(* Logix 5000 project; controller PBS_Perfusion vendor 1 type 14 code 217 rev 32.14; software revision 32.03; part 8 of 27 *)
(* tags used below, declared in another part *)
   Inp : BOOL;   // Alarm Condition Input 1=Alarm
   Inp_OoS : ALIAS FOR Com_AE.2;   // 1=Out of Service (from object's P_CmdSrc)
   Cfg_Exists : BOOL;   // 1=Alarm configured to exist, 0=Does not exist, don't scan
   Cfg_ResetReqd : BOOL;   // 1=Latched Alarm, a Reset is required to clear this Alarm
   Cfg_AckReqd : BOOL;   // 1=Acknowledge required for this Alarm
   Cfg_AllowShelve : BOOL;   // 1=Allow Operator to Shelve this Alarm
   Cfg_AllowDisable : BOOL;   // 1=Allow Maintenance to Disable this Alarm
   Cfg_Severity : DINT;   // Alarm Severity: 1..250=Low, 251..500=Medium, 501..750=High, 751..1000=Urgent
   Cfg_AlmMinOnT : DINT;   // Minimum time Alm output stays on (sec)
   PCfg_AllowExist : BOOL;   // 1=Alarm can be configured to exist, 0=other configs make alarm meaningless
   PCmd_Ack : BOOL;   // Program Command to Acknowledge alarm
   PCmd_Suppress : BOOL;   // Program Command to Suppress by Design (inhibits new alarm)
   PCmd_Unsuppress : BOOL;   // Program Command to Unsuppress (allows new alarm)
   PCmd_Unshelve : BOOL;   // Program Command to Unshelve (e.g., on shift change)
   Alm : ALIAS FOR Com_AE.0;   // Alarm output 1=In Alarm
   Ack : ALIAS FOR Com_AE.1;   // Alarm acknowledged status: 1=Ack rcvd
   Shelved : ALIAS FOR Com_AE.3;   // 1=Alarm has been Shelved by Operator (inhibits new alarm)
   Suppressed : ALIAS FOR Com_AE.6;   // 1=Alarm has been Suppressed by Program (inhibits new alarm)
   Disabled : ALIAS FOR Com_AE.9;   // 1=Alarm has been Disabled by Maintanance (inhibits new alarm)
   P_Alarm : BOOL;   // Unique Parameter Name for auto - discovery
   Wrk_Suppressed : BOOL;   // Internal Alarm Suppressed Status
   Com_AE : INT;   // Communication with HMI / Alarm/Event Server (see bit descriptions)
   OCmd_Unshelve : BOOL;   // Operator Command to Unshelve alarm (allows new alarm)
   OCmd_Shelve : BOOL;   // Operator Command to Shelve Alarm (inhibits new alarm)
   OCmd_Ack : BOOL;   // Operator Command to Acknowledge alarm
   MCmd_Enable : BOOL;   // Maintenance Command to Enable alarm (allows new alarm)
   MCmd_Disable : BOOL;   // Maintenance Command to Disable alarm (inhibits new alarm)
   ONS : DINT[3];
   REAL : DINT;
(* P_Alarm, continued *)

ROUTINE Prescan   (* ladder *)
// Clear "lurking" Commands
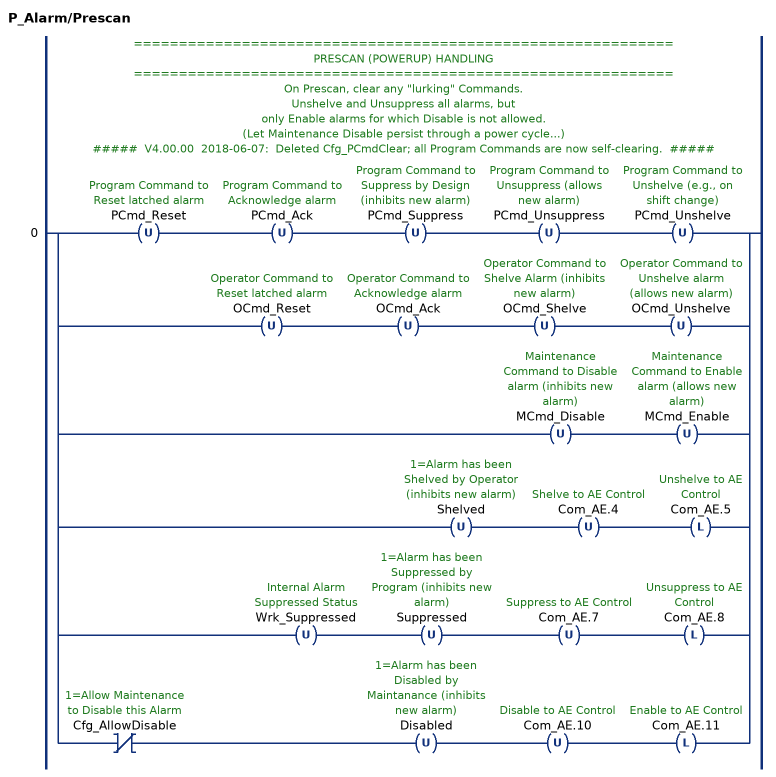
   // ============================================================
   // PRESCAN (POWERUP) HANDLING
   // ============================================================
   // On Prescan, clear any "lurking" Commands.
   // Unshelve and Unsuppress all alarms, but
   // only Enable alarms for which Disable is not allowed.
   // (Let Maintenance Disable persist through a power cycle...)
   // #####  V4.00.00  2018-06-07:  Deleted Cfg_PCmdClear; all Program Commands are now self-clearing.  #####
   0: [OTU(PCmd_Reset) OTU(PCmd_Ack) OTU(PCmd_Suppress) OTU(PCmd_Unsuppress) OTU(PCmd_Unshelve) ,OTU(OCmd_Reset) OTU(OCmd_Ack) OTU(OCmd_Shelve) OTU(OCmd_Unshelve) ,OTU(MCmd_Disable) OTU(MCmd_Enable) ,OTU(Shelved) OTU(Com_AE.4) OTL(Com_AE.5) ,OTU(Wrk_Suppressed) OTU(Suppressed) OTU(Com_AE.7) OTL(Com_AE.8) ,XIO(Cfg_AllowDisable) OTU(Disabled) OTU(Com_AE.10) OTL(Com_AE.11) ];
END_ROUTINE
END_ADD_ON_INSTRUCTION

ADD_ON_INSTRUCTION P_AOut   (* revision 4.10 .01 Release, vendor Rockwell Automation, ExecutePrescan, ExecuteEnableInFalse *)
// Analog Output
// Revision note:
// See Instruction Help for a summary of changes, and see 4.10 Release Notes for details.
// Help:
// Copyright © Rockwell Automation, Inc.  All Rights Reserved.
// This Instruction controls an Analog Output and provides:
// *  Program and Operator entry of target CV in Engineering Units
// *  Ramping of Output CV to target at specified Rate of Change (EU/sec)
// *  Clamping of Output CV at configured minimum and maximum limits
// *  Scaling of Output CV from Engineering Units to Raw (I/O card) Units
// *  Monitoring of Interlock conditions which cause output to shed
// *  Configurable shed to HOLD or to configured value
// *  Monitoring of I/O communication faults
// *  Alarms for Interlock Trip, I/O Fault
// *  "Available" status for use by automation logic to know whether Output
//       can be controlled by other objects.
// Command Sources are arbitrated by a P_CmdSrc Add-On Instruction instance.
// Command Sources: Operator, Program, External, Override, Maintenance, Out of
// Service, Hand.  Alarms are provided by P_Alarm Add-On Instruction instances.
// SUMMARY OF CHANGES FROM PREVIOUS VERSION (4.10.00)
// See 4.10 Release Notes for details.
// * No changes, uprevved because P_CmdSrc 4.10.01 is used.
// PREVIOUS VERSION (4.00.00)
// See 4.10 Release Notes for details.
// * Changed Sts_Available to use input availability from interlocks.
// * Updated to P_CmdSrc V4.10.00.
// * Added Cfg_HasMoreObj
// SUMMARY OF CHANGES FROM PREVIOUS VERSION (3.5-11)
// See 4.00 Release Notes for details.
// * Changed Inf_ items to HMI_, and added Cfg_Area for security.
// * Added notify and unack count rollup for associated object(s).
// * Changed "Mode" to "Command Source" using P_CmdSrc 4.00.00.
// * Deleted Cfg_PCmdClear; all Program Commands are now self-clearing.
// * Aligned ready bit naming with command bit names.
// * Added unacked alarm count.
// * Added  configurable decimal places for display on HMI.
// * Corrected CV Rate of Change Limiting when one direction is unlimited.
// * All OCmds/MCmds and ORdys/MRdys are now Local Tags.
// * Added Sts_RdyAck and Sts_RdyReset for use by external objects.
VAR_INPUT
   Inp_Tieback : REAL; {visible}   // Tieback CV (in raw, Out_CV units) used in Hand or Init
   Inp_IntlkOK : BOOL := 1; {visible}   // 1=Interlocks OK, Analog Output can be set
   Inp_NBIntlkOK : BOOL := 1; {visible}   // 1=Non-Bypassable Interlocks OK, Analog Output can be set
   Inp_IntlkAvail : BOOL;   // 1 = Interlock Availibility OK
   Inp_IOFault : BOOL;   // Input Communication Status 0=OK, 1=fail
   Inp_Sim : BOOL;   // 1=I/O are being simulated, set output CV to 0, ignore I/O Fault
   Inp_Hand : ALIAS FOR CmdSrc.Inp_Hand; {visible}
   Inp_Ovrd : ALIAS FOR CmdSrc.Inp_Ovrd; {visible}
   Inp_OvrdCV : REAL; {visible}   // CV target in Override Mode
   Inp_ExtInh : ALIAS FOR CmdSrc.Inp_ExtInh;
   Inp_Reset : BOOL;   // 1=Reset shed latches and cleared alarms
   Cfg_ShedHold : BOOL;   // 1=Hold Output on Interlock, 0=Go to Cfg_IntlkCV
   Cfg_SkipRoCLim : BOOL;   // 1=Skip RoC Limiting in Intlk, Maint, Ovrd
   Cfg_SetTrack : BOOL := 1;   // 1=PSets track OSets in Oper, OSets track PSets in Prog, 0=no tracking
   Cfg_SetTrackOvrdHand : BOOL;   // 1=Prog/Oper Settings track Override/Hand CV
   Cfg_HasIntlkObj : BOOL;   // 1=Tells HMI a P_Intlk is connected to Inp_Intlk
   Cfg_HasMoreObj : BOOL;   // 1=Tells HMI an object with more info is available
   Cfg_HasCVNav : BOOL;   // 1=Tells HMI to enable navigation to a connected CV object
   Cfg_OvrdIntlk : BOOL;   // 1=Override ignores Bypassable Intlk; 0=always use Intlk
   Cfg_ShedOnIOFault : BOOL := 1;   // 1=Stop Motor and Alarm on I/O Fault; 0=Alarm only on I/O Fault
   Cfg_DecPlcs : DINT := 2;   // Number of decimal places for CV display (0..6)
   Cfg_HasIntlkTripAlm : ALIAS FOR IntlkTrip.Cfg_Exists;   // 1=Interlock Trip Alarm exists and will be checked
   Cfg_HasIOFaultAlm : ALIAS FOR IOFault.Cfg_Exists;   // 1=I/O Fault Alarm exists and will be checked
   Cfg_IntlkTripResetReqd : ALIAS FOR IntlkTrip.Cfg_ResetReqd;   // 1=Reset required to clear Interlock Trip Alarm
   Cfg_IOFaultResetReqd : ALIAS FOR IOFault.Cfg_ResetReqd;   // 1=Reset required to clear I/O Fault Alarm
   Cfg_IntlkTripAckReqd : ALIAS FOR IntlkTrip.Cfg_AckReqd;   // 1=Acknowledge required for Interlock Trip Alarm
   Cfg_IOFaultAckReqd : ALIAS FOR IOFault.Cfg_AckReqd;   // 1=Acknowledge required for I/O Fault Alarm
   Cfg_IntlkTripSeverity : ALIAS FOR IntlkTrip.Cfg_Severity;   // Interlock Trip Alarm Severity: 1..250=Low, 251..500=Medium, 501..750=High, 751..1000=Urgent
   Cfg_IOFaultSeverity : ALIAS FOR IOFault.Cfg_Severity;   // I/O Fault Alarm Severity: 1..250=Low, 251..500=Medium, 501..750=High, 751..1000=Urgent
   Cfg_MinCV : REAL;   // Minimum CV (in EU, for limiting)
   Cfg_MaxCV : REAL := 100.0;   // Maximum CV (in EU, for limiting)
   Cfg_CVRoCLimInc : REAL;   // CV Rate of Change Limit, Increasing, (EU/sec, 0=unlimited)
   Cfg_CVRoCLimDec : REAL;   // CV Rate of Change Limit, Decreasing, (EU/sec, 0=unlimited)
   Cfg_IntlkCV : REAL;   // CV Target when interlocked (if not Cfg_ShedHold) (EU)
   Cfg_CVEUMin : REAL;   // CV Minimum in Engineering Units (for scaling)
   Cfg_CVEUMax : REAL := 100.0;   // CV Maximum in Engineering Units (for scaling)
   Cfg_CVRawMin : REAL;   // CV Minimum in I/O (raw) Units (for scaling)
   Cfg_CVRawMax : REAL := 100.0;   // CV Maximum in I/O (raw) Units (for scaling)
   Cfg_MaxInactiveCV : REAL;   // When Val_CVOut is greater than this value (in CV EU) set Sts_Active (for HMI)
   PSet_CV : REAL;   // Program Setting of Controlled Variable (output) (in EU)
   PSet_Owner : DINT;   // Program Owner Request ID (non-zero) or Release (zero)
   XSet_CV : REAL;   // External Setting of Controlled Variable (output) (in EU)
   PCmd_Prog : ALIAS FOR CmdSrc.PCmd_Prog;
   PCmd_Oper : ALIAS FOR CmdSrc.PCmd_Oper;
   PCmd_Lock : ALIAS FOR CmdSrc.PCmd_Lock;
   PCmd_Unlock : ALIAS FOR CmdSrc.PCmd_Unlock;
   PCmd_Normal : ALIAS FOR CmdSrc.PCmd_Normal;
   PCmd_Reset : BOOL;   // Program Command to reset shed latches and cleared alarms
   PCmd_IntlkTripAck : ALIAS FOR IntlkTrip.PCmd_Ack;   // Program Command to Acknowledge Interlock Trip Alarm
   PCmd_IntlkTripSuppress : ALIAS FOR IntlkTrip.PCmd_Suppress;   // Program Command to Suppress Interlock Trip Alarm
   PCmd_IntlkTripUnsuppress : ALIAS FOR IntlkTrip.PCmd_Unsuppress;   // Program Command to Unsuppress Interlock Trip Alarm
   PCmd_IntlkTripUnshelve : ALIAS FOR IntlkTrip.PCmd_Unshelve;   // Program Command to Unshelve Interlock Trip Alarm
   PCmd_IOFaultAck : ALIAS FOR IOFault.PCmd_Ack;   // Program Command to Acknowledge I/O Fault Alarm
   PCmd_IOFaultSuppress : ALIAS FOR IOFault.PCmd_Suppress;   // Program Command to Suppress I/O Fault Alarm
   PCmd_IOFaultUnsuppress : ALIAS FOR IOFault.PCmd_Unsuppress;   // Program Command to Unsuppress I/O Fault Alarm
   PCmd_IOFaultUnshelve : ALIAS FOR IOFault.PCmd_Unshelve;   // Program Command to Unshelve I/O Fault Alarm
   MCmd_Rel : ALIAS FOR CmdSrc.MCmd_Rel;
   OCmd_Unlock : ALIAS FOR CmdSrc.OCmd_Unlock;
   XCmd_Acq : ALIAS FOR CmdSrc.XCmd_Acq;
   XCmd_Rel : ALIAS FOR CmdSrc.XCmd_Rel;
   XCmd_Reset : BOOL;   // External Command to reset shed latches and cleared alarms
END_VAR
VAR_OUTPUT
   Out_CV : REAL; {access Read Only, visible}   // CV Output in Raw (I/O Card) Units
   Val_CVSet : REAL; {access Read Only, visible}   // Value of selected CV Setting (before rate limiting, in EU)
   Val_CVOut : REAL; {access Read Only, visible}   // Value of CV Output (after rate limiting) (in EU)
   Val_CVEUMin : REAL; {access Read Only}   // Minimum of scaled range = MIN (Cfg_CVEUMin, Cfg_CVEUMax)
   Val_CVEUMax : REAL := 100.0; {access Read Only}   // Maximum of scaled range = MAX (Cfg_CVEUMin, Cfg_CVEUMax)
   SrcQ_IO : DINT; {access Read Only}   // Source and Quality of primary I/O (enumeration)
   SrcQ : DINT; {access Read Only}   // Source and Quality of primary Val/Sts (enumeration)
   Val_Sts : DINT; {access Read Only}   // 0=AtTgt 1=RampDn 2=RampUp 3=ClampMin 4=ClampMax
   Val_Fault : DINT; {access Read Only}   // Device Fault Status 0=none, 32=I/OFault, 34=CfgErr
   Val_NotifyAll : DINT; {access Read Only}   // Highest Alarm prio and ack status this object + channel (enum)
   Val_UnackAlmC : DINT; {access Read Only}   // Count of Unacknowledged Alarms
   Val_Owner : DINT; {access Read Only}   // Current Object Owner ID (0=not owned)
   Sts_Ramping : BOOL; {access Read Only}   // 1=CV is ramping to target
   Sts_Clamped : BOOL; {access Read Only}   // 1=CV Set is clamped at CVMin or CVMax
   Sts_SkipRoCLim : BOOL; {access Read Only}   // 1=Rate of Change Limiting was skipped this scan (Maint, Ovrd, Intlk, Hand)
   Sts_Active : BOOL; {access Read Only}   // 1=CV is greater than Cfg_MaxInactiveCV, show graphic symbol as "active"
   Sts_Available : BOOL; {access Read Only}   // 1=Analog Output available for control by automation (Prog)
   Sts_Bypass : BOOL; {access Read Only}   // 1=Bypassable Interlocks are Bypassed
   Sts_BypActive : BOOL; {access Read Only}   // 1=Bypassing Active (Bypassed or Maintenance)
   Sts_NotRdy : BOOL; {access Read Only}   // 1=Device Not Ready, see detail bits for reason
   Nrdy_CfgErr : BOOL; {access Read Only}   // 1=Device Not Ready: Configuration Error
   Nrdy_Intlk : BOOL; {access Read Only}   // 1=Device Not Ready: Interlock Not OK
   Nrdy_IOFault : BOOL; {access Read Only}   // 1=Device Not Ready: I/O Fault (Shed Requires Reset)
   Nrdy_OoS : BOOL; {access Read Only}   // 1=Device Not Ready: Device is Out of Service
   Sts_MaintByp : BOOL; {access Read Only}   // 1=Device has a Maintenance Bypass function active
   Sts_AlmInh : BOOL; {access Read Only}   // 1=One or more Alarms Shelved, Disabled or Suppressed
   Sts_Err : BOOL; {access Read Only, visible}   // 1=Error in Config: see detail bits for reason
   Err_Limit : BOOL; {access Read Only}   // 1=Error in Config: CV Limits swapped
   Err_EU : BOOL; {access Read Only}   // 1=Error in Config: Scaled CV EU Min = Max
   Err_Raw : BOOL; {access Read Only}   // 1=Error in Config: Raw Output Scaling Min = Max
   Err_Alarm : BOOL; {access Read Only}   // 1=Error in Config: Alarm Min On Time, Shelf Time, Severity
   Sts_Hand : ALIAS FOR CmdSrc.Sts_Hand; {access Read Only, visible}
   Sts_OoS : ALIAS FOR CmdSrc.Sts_OoS; {access Read Only, visible}
   Sts_Maint : ALIAS FOR CmdSrc.Sts_Maint; {access Read Only, visible}
   Sts_Ovrd : ALIAS FOR CmdSrc.Sts_Ovrd; {access Read Only, visible}
   Sts_Ext : ALIAS FOR CmdSrc.Sts_Ext; {access Read Only, visible}
   Sts_Prog : ALIAS FOR CmdSrc.Sts_Prog; {access Read Only, visible}
   Sts_ProgLocked : ALIAS FOR CmdSrc.Sts_ProgLocked; {access Read Only}
   Sts_Oper : ALIAS FOR CmdSrc.Sts_Oper; {access Read Only, visible}
   Sts_OperLocked : ALIAS FOR CmdSrc.Sts_OperLocked; {access Read Only}
   Sts_Normal : ALIAS FOR CmdSrc.Sts_Normal; {access Read Only}
   Sts_ExtReqInh : ALIAS FOR CmdSrc.Sts_ExtReqInh; {access Read Only}
   Sts_ProgReqInh : ALIAS FOR CmdSrc.Sts_ProgReqInh; {access Read Only}
   Sts_MAcqRcvd : ALIAS FOR CmdSrc.Sts_MAcqRcvd; {access Read Only}
   Sts_RdyReset : ALIAS FOR ORdy_Reset; {access Read Only}   // 1=A latched alarm or shed condition is ready to be reset
   Sts_RdyAck : BOOL; {access Read Only}   // 1=An alarm is ready to be acknowledged
   Sts_IntlkTrip : ALIAS FOR IntlkTrip.Inp;   // 1=Status: CV held or forced by interlock NOT OK (1-shot)
   Alm_IntlkTrip : ALIAS FOR IntlkTrip.Alm;   // 1=Alarm: CV held or forced by interlock NOT OK
   Ack_IntlkTrip : ALIAS FOR IntlkTrip.Ack;   // 1=Interlock Trip Alarm has been acknowledged
   Sts_IntlkTripDisabled : ALIAS FOR IntlkTrip.Disabled;   // 1=Interlock Trip Alarm has been Disabled by Maintenance
   Sts_IntlkTripShelved : ALIAS FOR IntlkTrip.Shelved;   // 1=Interlock Trip Alarm has been Shelved by Operator
   Sts_IntlkTripSuppressed : ALIAS FOR IntlkTrip.Suppressed;   // 1=Interlock Trip Alarm has been Suppressed by Program
   Sts_IOFault : ALIAS FOR IOFault.Inp;   // 1=I/O Fault Status (0=OK, 1=Bad)
   Alm_IOFault : ALIAS FOR IOFault.Alm;   // 1=I/O Fault Alarm
   Ack_IOFault : ALIAS FOR IOFault.Ack;   // 1=I/O Fault Alarm has been acknowledged
   Sts_IOFaultDisabled : ALIAS FOR IOFault.Disabled;   // 1=I/O Fault Alarm has been Disabled by Maintenance
   Sts_IOFaultShelved : ALIAS FOR IOFault.Shelved;   // 1=I/O Fault Alarm has been Shelved by Operator
   Sts_IOFaultSuppressed : ALIAS FOR IOFault.Suppressed;   // 1=I/O Fault Alarm has been Suppressed by Program
   MRdy_Rel : ALIAS FOR CmdSrc.MRdy_Rel; {access Read Only}
   ORdy_Unlock : ALIAS FOR CmdSrc.ORdy_Unlock; {access Read Only}
   P_AOut : BOOL;   // Unique Parameter Name for auto - discovery
END_VAR
VAR
   CmdSrc : P_CmdSrc := (Cfg_HasOper := 1, Cfg_HasOperLocked := 1, Cfg_HasProg := 1, Cfg_HasProgLocked := 1, Cfg_HasMaint := 1, Cfg_HasMOoS := 1, Cfg_OvrdOverLock := 1, Sts_bSrc := 1);   // Control / Command Source Selection
   IOFault : P_Alarm := (Cfg_AckReqd := 1, Cfg_AllowShelve := 1, Cfg_AllowDisable := 1, Cfg_Severity := 1000, Cfg_AlmMinOnT := 5, PCfg_AllowExist := 1, Ack := 1);   // I/O Fault Alarm
   IntlkTrip : P_Alarm := (Cfg_AckReqd := 1, Cfg_AllowShelve := 1, Cfg_AllowDisable := 1, Cfg_Severity := 500, Cfg_AlmMinOnT := 5, PCfg_AllowExist := 1, Ack := 1);   // Interlock Trip Alarm
   Cfg_Tag : STRING_20 := 'P_AOut';   // Tagname for display on HMI
   Cfg_Label : STRING_20 := 'Analog Output';   // Label for graphic symbol displayed on HMI
   Cfg_Desc : STRING_40 := 'Analog Output';   // Description for display on HMI
   Wrk_Notify : DINT; {access None}   // Buffer for building Val_Notify
   Wrk_Bypass : BOOL; {access None}   // Internal Bypassable Interlocks are Bypassed flag
   Cfg_EU : STRING_8 := '%';   // Engineering Units for display on HMI
   Wrk_CV : REAL; {access None}   // Working copy of Speed Reference (for limiting)
   Wrk_CVSet : REAL; {access None}   // Final selected CV to feed to RoC Limiter
   Wrk_CVOut : REAL; {access None}   // Wroking value of CV after Rate Limiting
   Wrk_IntlkTripONS : BOOL; {access None}   // Interlock Tripped This Scan
   Wrk_ScanTime : REAL; {access None}   // Seconds since previous scan
   Wrk_StepInc : REAL; {access None}   // Amount to change CVOut this scan for increase rate limiting
   Wrk_ScanT : TIMER := (PRE := 2147483647); {access None}   // Scan Timer (milliseconds, always runs)
   Wrk_SelCVDINT : DINT; {access None}   // Selected CV check for Infinite or Non A Number
   HMI_Tab : SINT;   // Tab to display (FTView ME)
   Val_Notify : SINT; {access Read Only}   // Current Alarm Level and Acknowledgement (enumeration)
   Wrk_Sts : DINT; {access None}   // Buffer for building Val_Sts
   Wrk_Fault : DINT; {access None}   // Buffer for building Val_Fault
   Wrk_SrcQ : DINT; {access None}   // Register for building Source / Quality enumeration
   HMI_Type : STRING_16 := 'P_AOut'; {access Read Only}   // Must contain AOI name, used for HMI and Information S/W
   Wrk_StepDec : REAL; {access None}   // Amount to change CVOut this scan for decrease rate limiting
   HMI_Lib : STRING_12 := 'RA-BAS'; {access Read Only}   // Display Library for Faceplate call-up
   Cfg_CVNavTag : STRING_NavTag;   // Tagname for destination of CV Navigation button
   Wrk_ShedIntlkCV : BOOL; {access None}   // Output CV being held at Interlock value
   Wrk_ShedHold : BOOL; {access None}   // Output CV being held at last good value
   Cfg_Area : STRING_Area := 'area01';   // Process Area for security
   Wrk_UnackAlmC : DINT; {access None}   // Buffer for building Val_UnackAlmC
   ORdy_CV : BOOL; {access Read Only}   // 1=Ready for OSet_CV (enables data entry field)
   ORdy_ResetAckAll : BOOL; {access Read Only}   // 1=Ready for OCmd_ResetAckAll (enables HMI button)
   ORdy_Reset : BOOL; {access Read Only}   // 1=Ready for OCmd_Reset (enables HMI button)
   MRdy_Check : BOOL; {access Read Only}   // 1=Ready for MCmd_Check (enables HMI button)
   MRdy_Bypass : BOOL; {access Read Only}   // 1=Ready for MCmd_Bypass (enables HMI button)
   OCmd_ResetAckAll : BOOL;   // Operator Command to Reset all Alarms and latched Shed conditions
   OCmd_Reset : BOOL;   // Oper Cmd to reset shed latches and cleared alarms
   MCmd_Check : BOOL;   // Maintenance Command to Check (not bypass) all Interlocks
   MCmd_Bypass : BOOL;   // Maintenance Command to Bypass all Bypassable Interlocks
   OSet_CV : REAL;   // Operator Setting of Controlled Variable (output) (in EU)
END_VAR

ROUTINE EnableInFalse   (* ladder *)
// Out of Service is asserted, Output OFF (zero), Alarms inhibited.
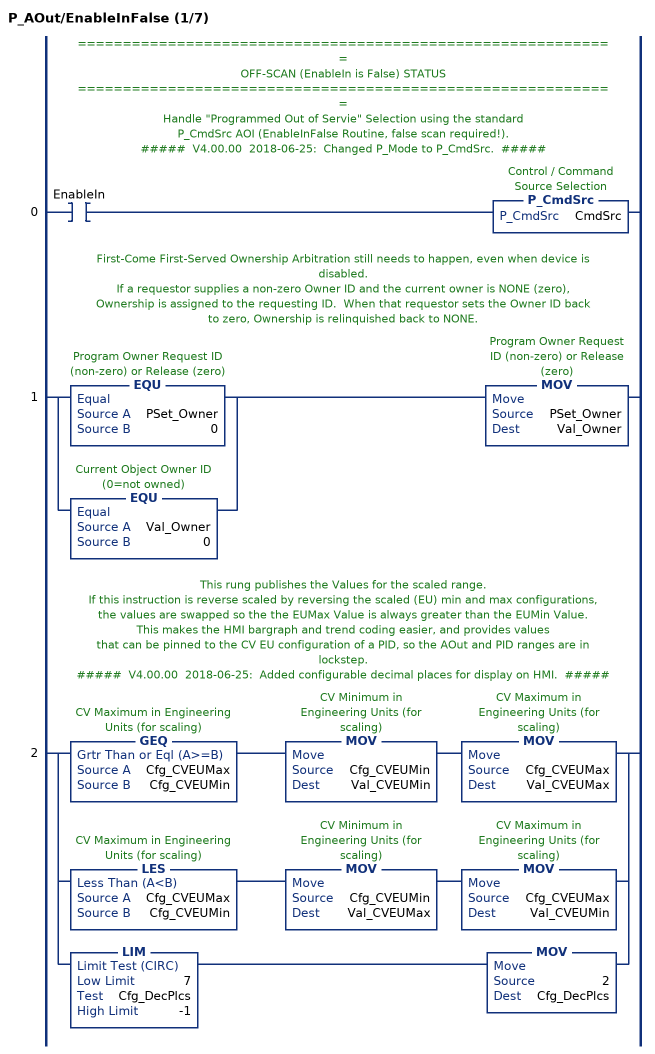
   // ============================================================
   // OFF-SCAN (EnableIn is False) STATUS
   // ============================================================
   // Handle "Programmed Out of Servie" Selection using the standard
   // P_CmdSrc AOI (EnableInFalse Routine, false scan required!).
   // #####  V4.00.00  2018-06-25:  Changed P_Mode to P_CmdSrc.  #####
   0: XIC(EnableIn)P_CmdSrc(CmdSrc);
   // First-Come First-Served Ownership Arbitration still needs to happen, even when device is disabled.
   // If a requestor supplies a non-zero Owner ID and the current owner is NONE (zero),
   // Ownership is assigned to the requesting ID.  When that requestor sets the Owner ID back
   // to zero, Ownership is relinquished back to NONE.
   1: [EQU(PSet_Owner,0) ,EQU(Val_Owner,0) ]MOV(PSet_Owner,Val_Owner);
   // This rung publishes the Values for the scaled range.
   // If this instruction is reverse scaled by reversing the scaled (EU) min and max configurations,
   // the values are swapped so the the EUMax Value is always greater than the EUMin Value.
   // This makes the HMI bargraph and trend coding easier, and provides values
   // that can be pinned to the CV EU configuration of a PID, so the AOut and PID ranges are in lockstep.
   // #####  V4.00.00  2018-06-25:  Added configurable decimal places for display on HMI.  #####
   2: [GEQ(Cfg_CVEUMax,Cfg_CVEUMin) MOV(Cfg_CVEUMin,Val_CVEUMin) MOV(Cfg_CVEUMax,Val_CVEUMax) ,LES(Cfg_CVEUMax,Cfg_CVEUMin) MOV(Cfg_CVEUMin,Val_CVEUMax) MOV(Cfg_CVEUMax,Val_CVEUMin) ,LIM(7,Cfg_DecPlcs,-1) MOV(2,Cfg_DecPlcs) ];
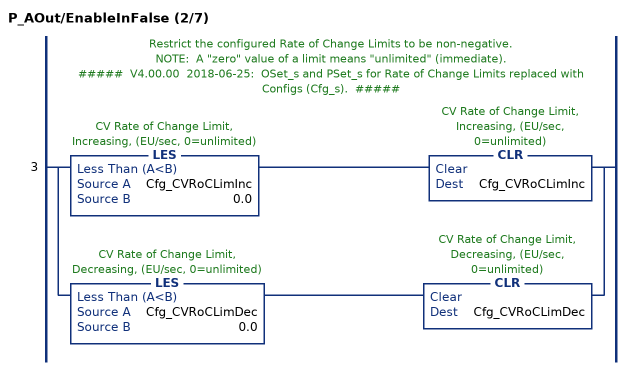
   // Restrict the configured Rate of Change Limits to be non-negative.
   // NOTE:  A "zero" value of a limit means "unlimited" (immediate).
   // #####  V4.00.00  2018-06-25:  OSet_s and PSet_s for Rate of Change Limits replaced with Configs (Cfg_s).  #####
   3: [LES(Cfg_CVRoCLimInc,0.0) CLR(Cfg_CVRoCLimInc) ,LES(Cfg_CVRoCLimDec,0.0) CLR(Cfg_CVRoCLimDec) ];
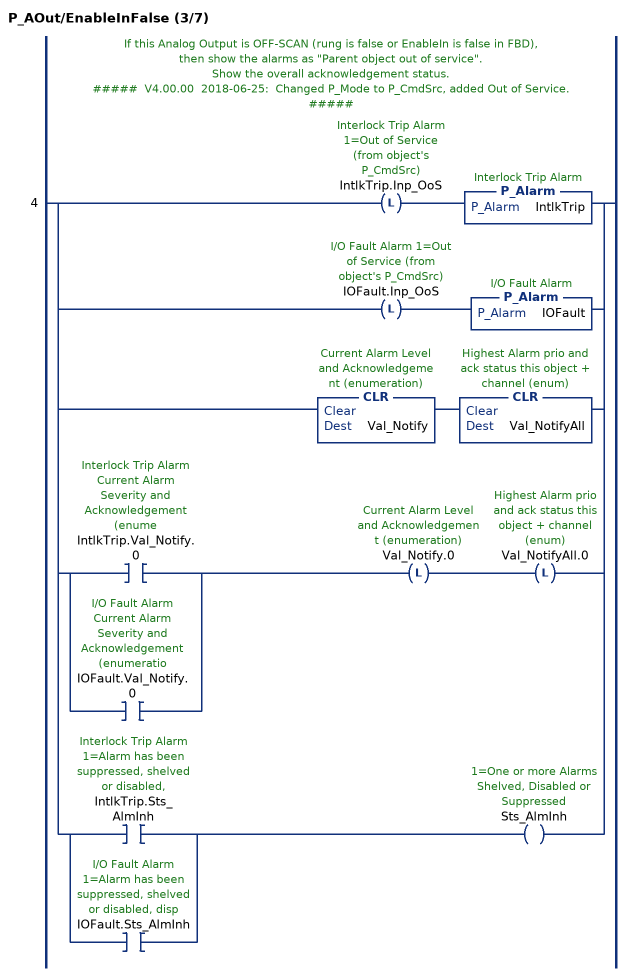
   // If this Analog Output is OFF-SCAN (rung is false or EnableIn is false in FBD),
   // then show the alarms as "Parent object out of service".
   // Show the overall acknowledgement status.
   // #####  V4.00.00  2018-06-25:  Changed P_Mode to P_CmdSrc, added Out of Service.  #####
   4: [OTL(IntlkTrip.Inp_OoS) P_Alarm(IntlkTrip) ,OTL(IOFault.Inp_OoS) P_Alarm(IOFault) ,CLR(Val_Notify) CLR(Val_NotifyAll) ,[XIC(IntlkTrip.Val_Notify.0) ,XIC(IOFault.Val_Notify.0) ] OTL(Val_Notify.0) OTL(Val_NotifyAll.0) ,[XIC(IntlkTrip.Sts_AlmInh) ,XIC(IOFault.Sts_AlmInh) ] OTE(Sts_AlmInh) ];
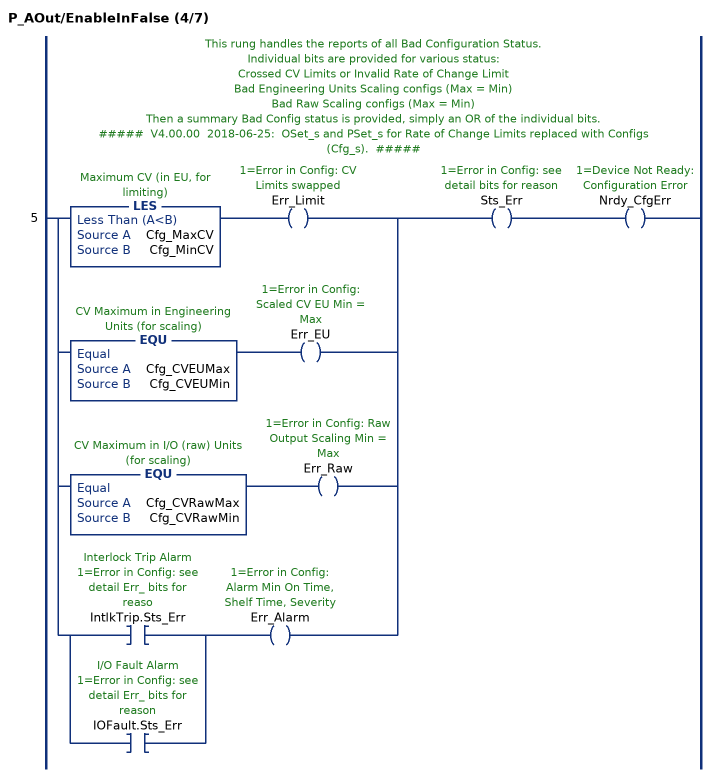
   // This rung handles the reports of all Bad Configuration Status.
   // Individual bits are provided for various status:
   // Crossed CV Limits or Invalid Rate of Change Limit
   // Bad Engineering Units Scaling configs (Max = Min)
   // Bad Raw Scaling configs (Max = Min)
   // Then a summary Bad Config status is provided, simply an OR of the individual bits.
   // #####  V4.00.00  2018-06-25:  OSet_s and PSet_s for Rate of Change Limits replaced with Configs (Cfg_s).  #####
   5: [LES(Cfg_MaxCV,Cfg_MinCV) OTE(Err_Limit) ,EQU(Cfg_CVEUMax,Cfg_CVEUMin) OTE(Err_EU) ,EQU(Cfg_CVRawMax,Cfg_CVRawMin) OTE(Err_Raw) ,[XIC(IntlkTrip.Sts_Err) ,XIC(IOFault.Sts_Err) ] OTE(Err_Alarm) ]OTE(Sts_Err)OTE(Nrdy_CfgErr);
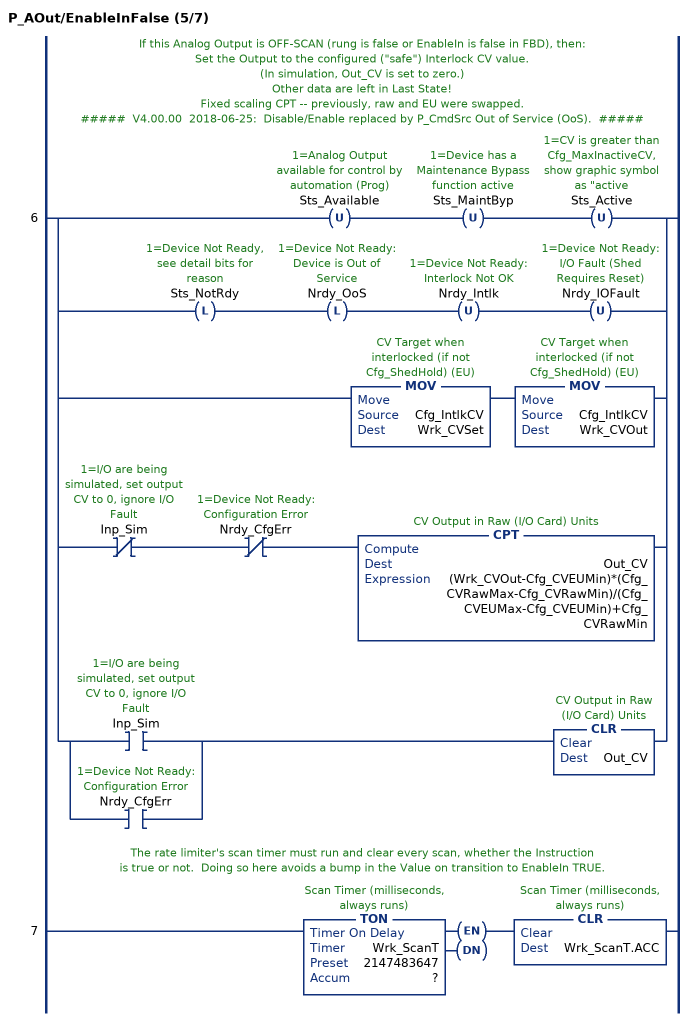
   // If this Analog Output is OFF-SCAN (rung is false or EnableIn is false in FBD), then:
   // Set the Output to the configured ("safe") Interlock CV value.
   // (In simulation, Out_CV is set to zero.)
   // Other data are left in Last State!
   // Fixed scaling CPT -- previously, raw and EU were swapped.
   // #####  V4.00.00  2018-06-25:  Disable/Enable replaced by P_CmdSrc Out of Service (OoS).  #####
   6: [OTU(Sts_Available) OTU(Sts_MaintByp) OTU(Sts_Active) ,OTL(Sts_NotRdy) OTL(Nrdy_OoS) OTU(Nrdy_Intlk) OTU(Nrdy_IOFault) ,MOV(Cfg_IntlkCV,Wrk_CVSet) MOV(Cfg_IntlkCV,Wrk_CVOut) ,XIO(Inp_Sim) XIO(Nrdy_CfgErr) CPT(Out_CV,(Wrk_CVOut-Cfg_CVEUMin)*(Cfg_CVRawMax-Cfg_CVRawMin)/(Cfg_CVEUMax-Cfg_CVEUMin)+Cfg_CVRawMin) ,[XIC(Inp_Sim) ,XIC(Nrdy_CfgErr) ] CLR(Out_CV) ];
   // The rate limiter's scan timer must run and clear every scan, whether the Instruction
   // is true or not.  Doing so here avoids a bump in the Value on transition to EnableIn TRUE.
   7: TON(Wrk_ScanT,?,?)CLR(Wrk_ScanT.ACC);
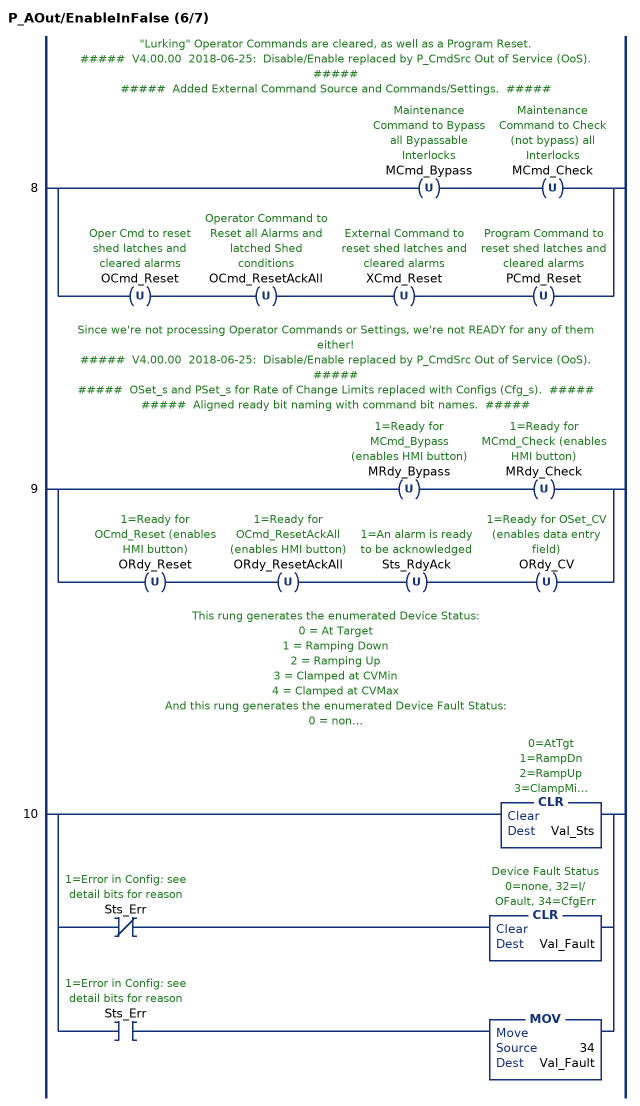
   // "Lurking" Operator Commands are cleared, as well as a Program Reset.
   // #####  V4.00.00  2018-06-25:  Disable/Enable replaced by P_CmdSrc Out of Service (OoS).  #####
   // #####  Added External Command Source and Commands/Settings.  #####
   8: [OTU(MCmd_Bypass) OTU(MCmd_Check) ,OTU(OCmd_Reset) OTU(OCmd_ResetAckAll) OTU(XCmd_Reset) OTU(PCmd_Reset) ];
   // Since we're not processing Operator Commands or Settings, we're not READY for any of them either!
   // #####  V4.00.00  2018-06-25:  Disable/Enable replaced by P_CmdSrc Out of Service (OoS).  #####
   // #####  OSet_s and PSet_s for Rate of Change Limits replaced with Configs (Cfg_s).  #####
   // #####  Aligned ready bit naming with command bit names.  #####
   9: [OTU(MRdy_Bypass) OTU(MRdy_Check) ,OTU(ORdy_Reset) OTU(ORdy_ResetAckAll) OTU(Sts_RdyAck) OTU(ORdy_CV) ];
   // This rung generates the enumerated Device Status:
   // 0 = At Target
   // 1 = Ramping Down
   // 2 = Ramping Up
   // 3 = Clamped at CVMin
   // 4 = Clamped at CVMax
   // And this rung generates the enumerated Device Fault Status:
   // 0 = none
   // 32 = I/O Fault
   // 34 = Configuration Error
   // #####  V4.00.00  2018-06-25:  Disable/Enable replaced by P_CmdSrc Out of Service (OoS).  #####
   10: [CLR(Val_Sts) ,XIO(Sts_Err) CLR(Val_Fault) ,XIC(Sts_Err) MOV(34,Val_Fault) ];
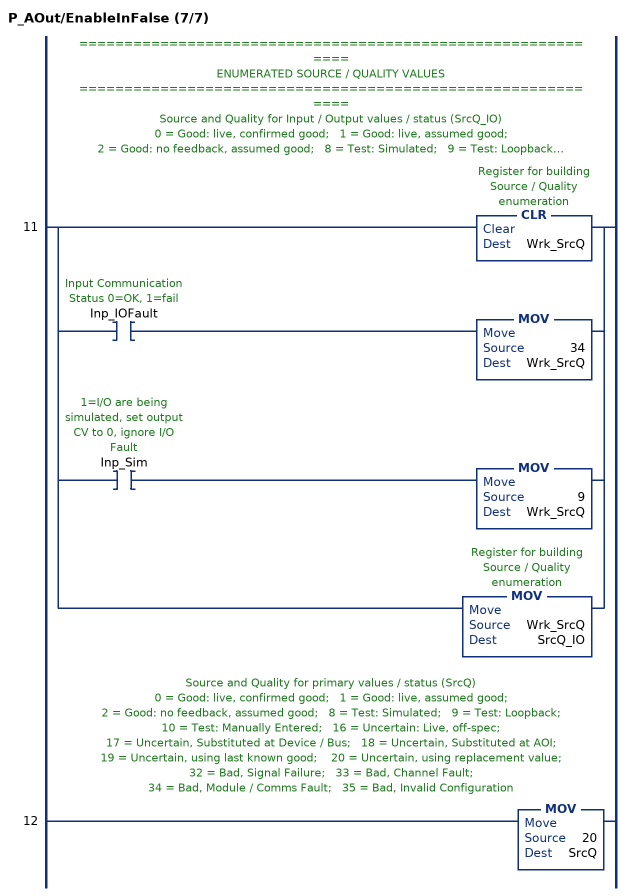
   // ============================================================
   // ENUMERATED SOURCE / QUALITY VALUES
   // ============================================================
   // Source and Quality for Input / Output values / status (SrcQ_IO)
   // 0 = Good: live, confirmed good;   1 = Good: live, assumed good;
   // 2 = Good: no feedback, assumed good;   8 = Test: Simulated;   9 = Test: Loopback;
   // 10 = Test: Manually Entered;   16 = Uncertain: Live, off-spec;
   // 17 = Uncertain, Substituted at Device / Bus;   18 = Uncertain, Substituted at AOI;
   // 19 = Uncertain, using last known good;    20 = Uncertain, using replacement value;
   // 32 = Bad, Signal Failure;   33 = Bad, Channel Fault;
   // 34 = Bad, Module / Comms Fault;   35 = Bad, Invalid Configuration
   11: [CLR(Wrk_SrcQ) ,XIC(Inp_IOFault) MOV(34,Wrk_SrcQ) ,XIC(Inp_Sim) MOV(9,Wrk_SrcQ) ,MOV(Wrk_SrcQ,SrcQ_IO) ];
   // Source and Quality for primary values / status (SrcQ)
   // 0 = Good: live, confirmed good;   1 = Good: live, assumed good;
   // 2 = Good: no feedback, assumed good;   8 = Test: Simulated;   9 = Test: Loopback;
   // 10 = Test: Manually Entered;   16 = Uncertain: Live, off-spec;
   // 17 = Uncertain, Substituted at Device / Bus;   18 = Uncertain, Substituted at AOI;
   // 19 = Uncertain, using last known good;    20 = Uncertain, using replacement value;
   // 32 = Bad, Signal Failure;   33 = Bad, Channel Fault;
   // 34 = Bad, Module / Comms Fault;   35 = Bad, Invalid Configuration
   12: MOV(20,SrcQ);
END_ROUTINE

ROUTINE Logic   (* ladder *)
// Normal Scan: control Analog Output
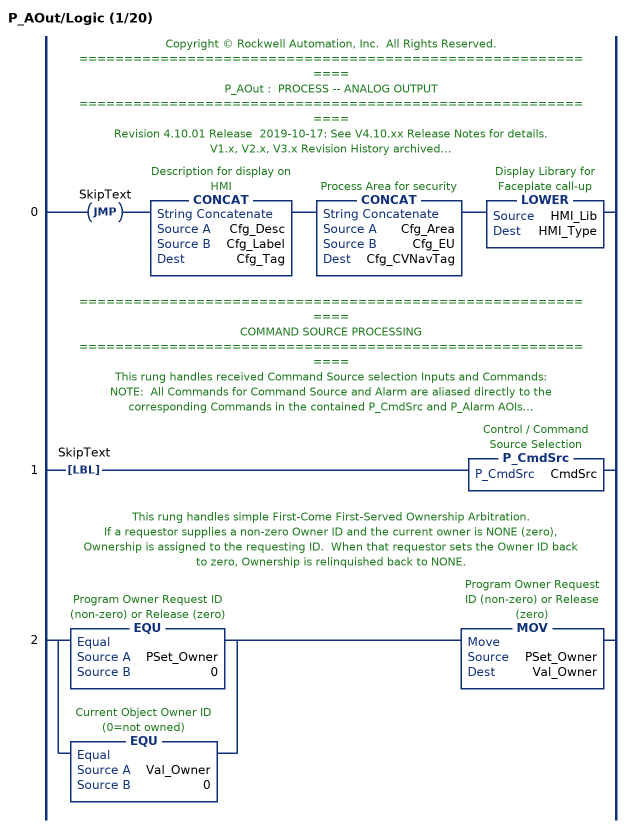
   // Copyright © Rockwell Automation, Inc.  All Rights Reserved.
   // ============================================================
   // P_AOut :  PROCESS -- ANALOG OUTPUT
   // ============================================================
   // Revision 4.10.01 Release  2019-10-17: See V4.10.xx Release Notes for details.
   // V1.x, V2.x, V3.x Revision History archived.
   // V4.00.00  2018-06-25:  Changed "Mode" to "Command Source". Changed Inf_items to HMI_,
   // and added Cfg_Area for security. Added unacked alarm count.
   // Deleted Cfg_PCmdClear; all Program Commands are now self-clearing.
   // Added  configurable decimal places for display on HMI.
   // Corrected CV Rate of Change Limiting when one direction is unlimited.
   // Aligned ready bit naming with command bit names.
   // All OCmds/MCmds and ORdys/MRdys are now Local Tags.
   // Added Sts_RdyAck and Sts_ResetReqd for use by external objects.
   // V4.10.00  2019-03-08:  Changed availability to use input availability from interlocks.
   // Updated to P_CmdSrc V4.10.00. Added Cfg_HasMoreObj.
   // V4.10.01  2019-10-17:  No changes, uprevved because P_CmdSrc 4.10.01 is used.
   // ============================================================
   // This Instruction controls an Analog Output and provides:
   // *  Program and Operator entry of target CV in Engineering Units
   // *  Ramping of Output CV to target at specified Rate of Change (EU/sec)
   // *  Clamping of Output CV at configured minimum and maximum limits
   // *  Scaling of Output CV from Engineering Units to Raw (I/O card) Units
   // *  Monitoring of Interlock conditions which cause output to shed
   // *  Configurable shed to HOLD or to configured SAFE value
   // *  Monitoring of I/O communication faults
   // *  Alarms for Interlock Trip, I/O Fault
   // *  "Available" status for use by automation logic to know whether Output
   //       can be controlled by other objects.
   // Command Sources are arbitrated by a P_CmdSrc Add-On Instruction instance.
   // Command Sources: Operator, Program, External, Override, Maintenance, Out of
   // Service, Hand.  Alarms are provided by P_Alarm Add-On Instruction instances.
   // ============================================================
   // SHOW LOCAL STRINGS
   // ============================================================
   // The STRINGs containing the text associated with each instance of this
   // instruction cannot be Input or Output Parameters, because STRINGs are not
   //  'atomic' types. (Inputs and Outputs must be SINT, INT, DINT, REAL, or BOOL.)
   // In order to make it easier to find and configure these STRINGs, this rung
   // was added.  THE JMP (and the LBL on the following rung)
   // MUST NOT BE REMOVED!!!
   // To view the STRINGs, go to the instruction instance (in LD or FBD), RIGHT-click
   // to bring up the context menu and select "Open Instruction Logic".
   // This rung will appear with the STRING values for the selected instance.
   // You may double-click the STRING values here to modify them as well.
   // #####  V4.00.00  2018-06-25:  Added string for Cfg_Area, renamed Inf_* to HMI_*.  #####
   0: JMP(SkipText)CONCAT(Cfg_Desc,Cfg_Label,Cfg_Tag)CONCAT(Cfg_Area,Cfg_EU,Cfg_CVNavTag)LOWER(HMI_Lib,HMI_Type);
   // ============================================================
   // COMMAND SOURCE PROCESSING
   // ============================================================
   // This rung handles received Command Source selection Inputs and Commands:
   // NOTE:  All Commands for Command Source and Alarm are aliased directly to the
   // corresponding Commands in the contained P_CmdSrc and P_Alarm AOIs.
   // #####  V4.00.00  2018-06-25:  Changed P_Mode to P_CmdSrc.  #####
   1: LBL(SkipText)P_CmdSrc(CmdSrc);
   // This rung handles simple First-Come First-Served Ownership Arbitration.
   // If a requestor supplies a non-zero Owner ID and the current owner is NONE (zero),
   // Ownership is assigned to the requesting ID.  When that requestor sets the Owner ID back
   // to zero, Ownership is relinquished back to NONE.
   2: [EQU(PSet_Owner,0) ,EQU(Val_Owner,0) ]MOV(PSet_Owner,Val_Owner);
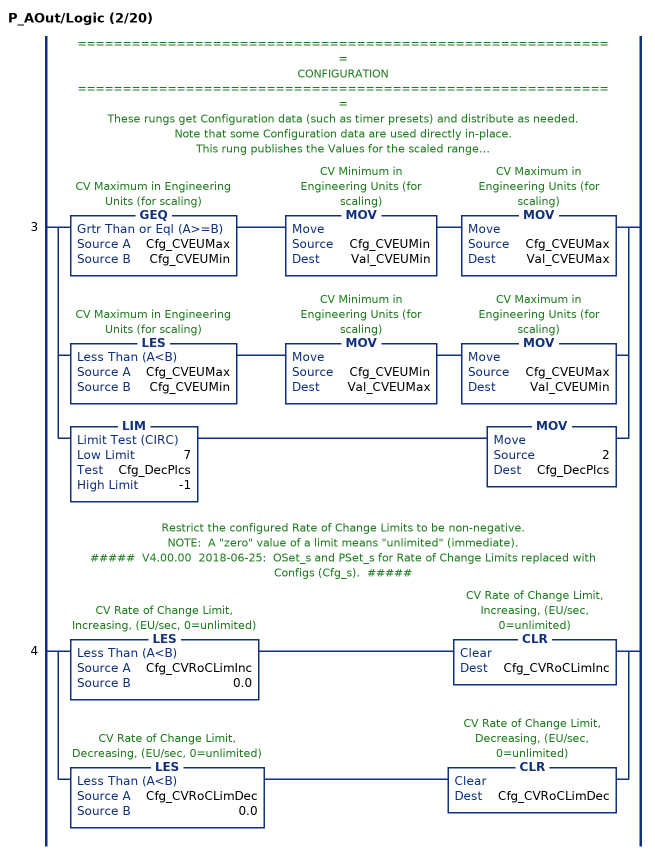
   // ============================================================
   // CONFIGURATION
   // ============================================================
   // These rungs get Configuration data (such as timer presets) and distribute as needed.
   // Note that some Configuration data are used directly in-place.
   // This rung publishes the Values for the scaled range.
   // If this instruction is reverse scaled by reversing the scaled (EU) min and max configurations,
   // the values are swapped so the the EUMax Value is always greater than the EUMin Value.
   // This makes the HMI bargraph and trend coding easier, and provides values
   // that can be pinned to the CV EU configuration of a PID, so the AOut and PID ranges are in lockstep.
   // #####  V4.00.00  2018-06-25:  Added configurable decimal places for display on HMI.  #####
   3: [GEQ(Cfg_CVEUMax,Cfg_CVEUMin) MOV(Cfg_CVEUMin,Val_CVEUMin) MOV(Cfg_CVEUMax,Val_CVEUMax) ,LES(Cfg_CVEUMax,Cfg_CVEUMin) MOV(Cfg_CVEUMin,Val_CVEUMax) MOV(Cfg_CVEUMax,Val_CVEUMin) ,LIM(7,Cfg_DecPlcs,-1) MOV(2,Cfg_DecPlcs) ];
   // Restrict the configured Rate of Change Limits to be non-negative.
   // NOTE:  A "zero" value of a limit means "unlimited" (immediate).
   // #####  V4.00.00  2018-06-25:  OSet_s and PSet_s for Rate of Change Limits replaced with Configs (Cfg_s).  #####
   4: [LES(Cfg_CVRoCLimInc,0.0) CLR(Cfg_CVRoCLimInc) ,LES(Cfg_CVRoCLimDec,0.0) CLR(Cfg_CVRoCLimDec) ];
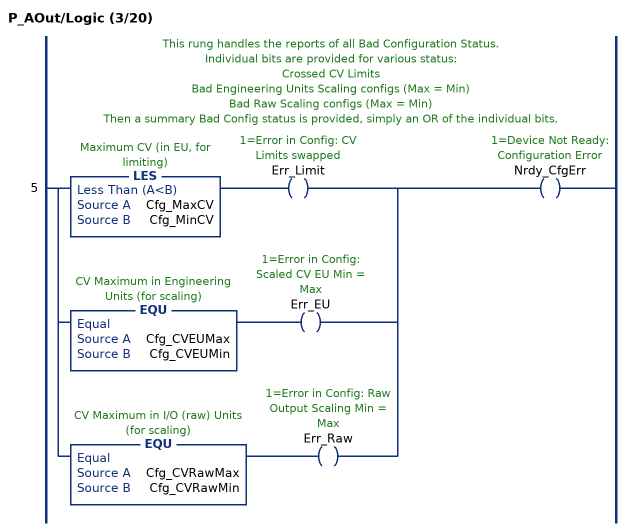
   // This rung handles the reports of all Bad Configuration Status.
   // Individual bits are provided for various status:
   // Crossed CV Limits
   // Bad Engineering Units Scaling configs (Max = Min)
   // Bad Raw Scaling configs (Max = Min)
   // Then a summary Bad Config status is provided, simply an OR of the individual bits.
   5: [LES(Cfg_MaxCV,Cfg_MinCV) OTE(Err_Limit) ,EQU(Cfg_CVEUMax,Cfg_CVEUMin) OTE(Err_EU) ,EQU(Cfg_CVRawMax,Cfg_CVRawMin) OTE(Err_Raw) ]OTE(Nrdy_CfgErr);
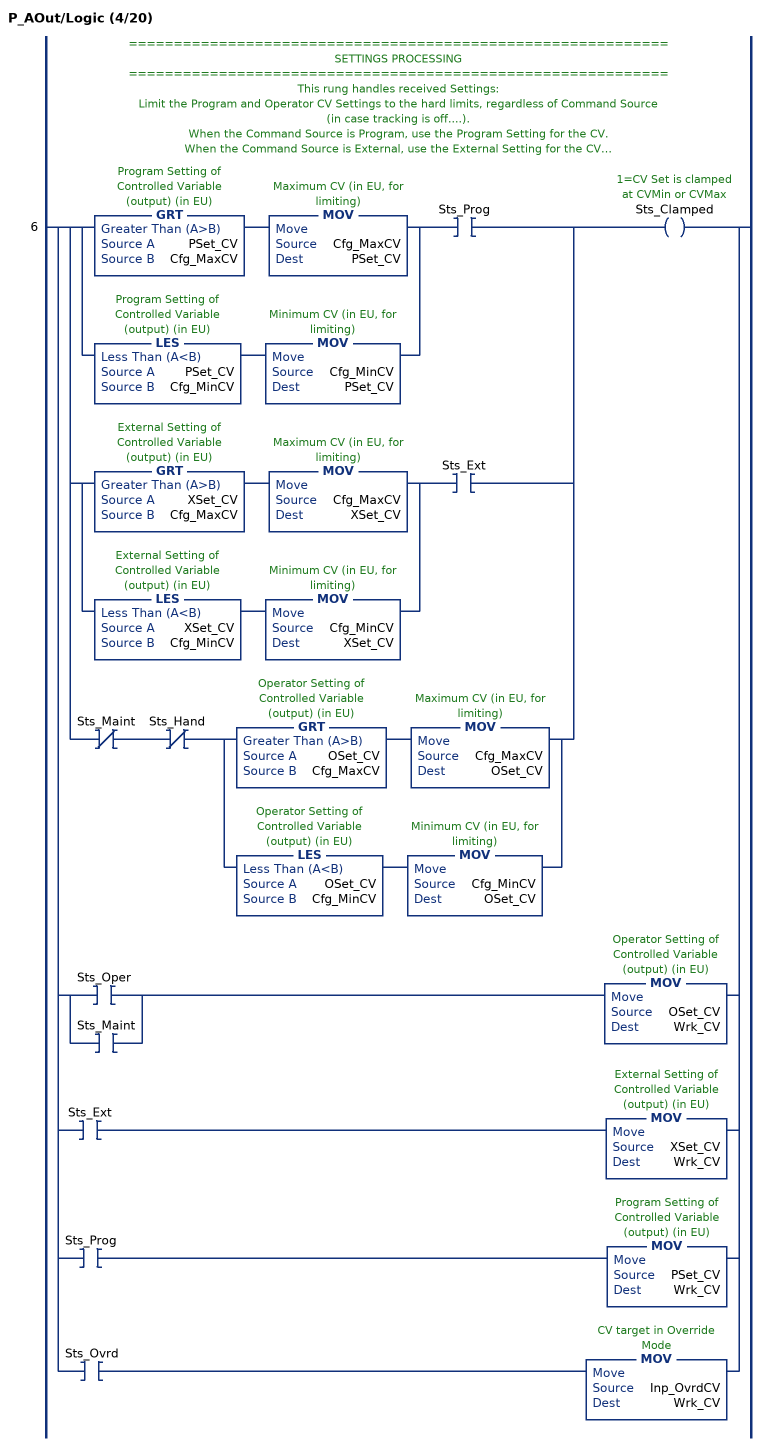
   // ============================================================
   // SETTINGS PROCESSING
   // ============================================================
   // This rung handles received Settings:
   // Limit the Program and Operator CV Settings to the hard limits, regardless of Command Source
   // (in case tracking is off....).
   // When the Command Source is Program, use the Program Setting for the CV.
   // When the Command Source is External, use the External Setting for the CV.
   // When the Command Source is Operator or Maintenance, use the Operator Setting.
   // When the Command Source is Override, use the Override CV input for the CV.
   // #####  V4.00.00  2018-06-25:  Added External Command Source and Commands/Settings.  #####
   6: [[[GRT(PSet_CV,Cfg_MaxCV) MOV(Cfg_MaxCV,PSet_CV) ,LES(PSet_CV,Cfg_MinCV) MOV(Cfg_MinCV,PSet_CV) ] XIC(Sts_Prog) ,[GRT(XSet_CV,Cfg_MaxCV) MOV(Cfg_MaxCV,XSet_CV) ,LES(XSet_CV,Cfg_MinCV) MOV(Cfg_MinCV,XSet_CV) ] XIC(Sts_Ext) ,XIO(Sts_Maint) XIO(Sts_Hand) [GRT(OSet_CV,Cfg_MaxCV) MOV(Cfg_MaxCV,OSet_CV) ,LES(OSet_CV,Cfg_MinCV) MOV(Cfg_MinCV,OSet_CV) ] ] OTE(Sts_Clamped) ,[XIC(Sts_Oper) ,XIC(Sts_Maint) ] MOV(OSet_CV,Wrk_CV) ,XIC(Sts_Ext) MOV(XSet_CV,Wrk_CV) ,XIC(Sts_Prog) MOV(PSet_CV,Wrk_CV) ,XIC(Sts_Ovrd) MOV(Inp_OvrdCV,Wrk_CV) ];
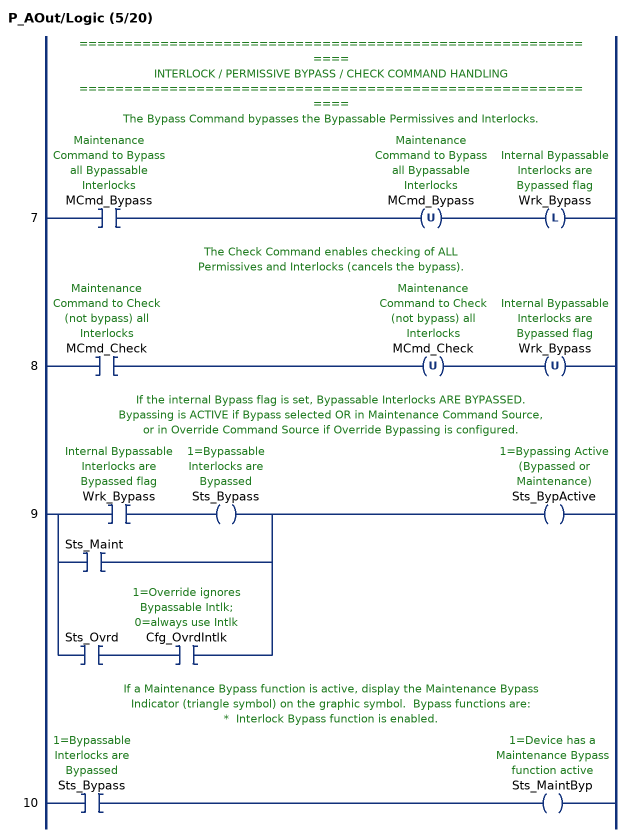
   // ============================================================
   // INTERLOCK / PERMISSIVE BYPASS / CHECK COMMAND HANDLING
   // ============================================================
   // The Bypass Command bypasses the Bypassable Permissives and Interlocks.
   7: XIC(MCmd_Bypass)OTU(MCmd_Bypass)OTL(Wrk_Bypass);
   // The Check Command enables checking of ALL
   // Permissives and Interlocks (cancels the bypass).
   8: XIC(MCmd_Check)OTU(MCmd_Check)OTU(Wrk_Bypass);
   // If the internal Bypass flag is set, Bypassable Interlocks ARE BYPASSED.
   // Bypassing is ACTIVE if Bypass selected OR in Maintenance Command Source,
   // or in Override Command Source if Override Bypassing is configured.
   9: [XIC(Wrk_Bypass) OTE(Sts_Bypass) ,XIC(Sts_Maint) ,XIC(Sts_Ovrd) XIC(Cfg_OvrdIntlk) ]OTE(Sts_BypActive);
   // If a Maintenance Bypass function is active, display the Maintenance Bypass
   // Indicator (triangle symbol) on the graphic symbol.  Bypass functions are:
   // *  Interlock Bypass function is enabled.
   10: XIC(Sts_Bypass)OTE(Sts_MaintByp);
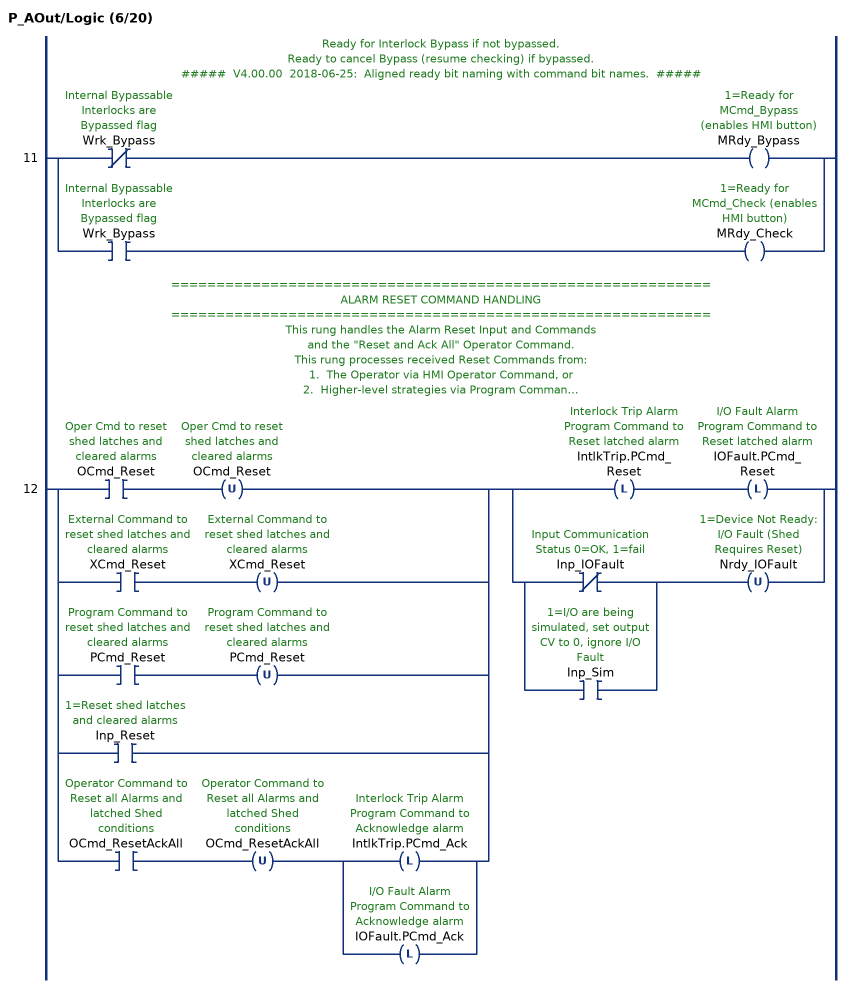
   // Ready for Interlock Bypass if not bypassed.
   // Ready to cancel Bypass (resume checking) if bypassed.
   // #####  V4.00.00  2018-06-25:  Aligned ready bit naming with command bit names.  #####
   11: [XIO(Wrk_Bypass) OTE(MRdy_Bypass) ,XIC(Wrk_Bypass) OTE(MRdy_Check) ];
   // ============================================================
   // ALARM RESET COMMAND HANDLING
   // ============================================================
   // This rung handles the Alarm Reset Input and Commands
   // and the "Reset and Ack All" Operator Command.
   // This rung processes received Reset Commands from:
   // 1.  The Operator via HMI Operator Command, or
   // 2.  Higher-level strategies via Program Command
   // 3.  Pushbuttons or other block via Input
   // and forwards the Reset to ALL Alarms and latched Shed conditions.
   // #####  V4.00.00  2018-06-25:  Deleted Cfg_PCmdClear; all Program Commands are now self-clearing.  #####
   // #####  Added External Command Source and Commands/Settings.  #####
   12: [XIC(OCmd_Reset) OTU(OCmd_Reset) ,XIC(XCmd_Reset) OTU(XCmd_Reset) ,XIC(PCmd_Reset) OTU(PCmd_Reset) ,XIC(Inp_Reset) ,XIC(OCmd_ResetAckAll) OTU(OCmd_ResetAckAll) [OTL(IntlkTrip.PCmd_Ack) ,OTL(IOFault.PCmd_Ack) ] ][OTL(IntlkTrip.PCmd_Reset) OTL(IOFault.PCmd_Reset) ,[XIO(Inp_IOFault) ,XIC(Inp_Sim) ] OTU(Nrdy_IOFault) ];
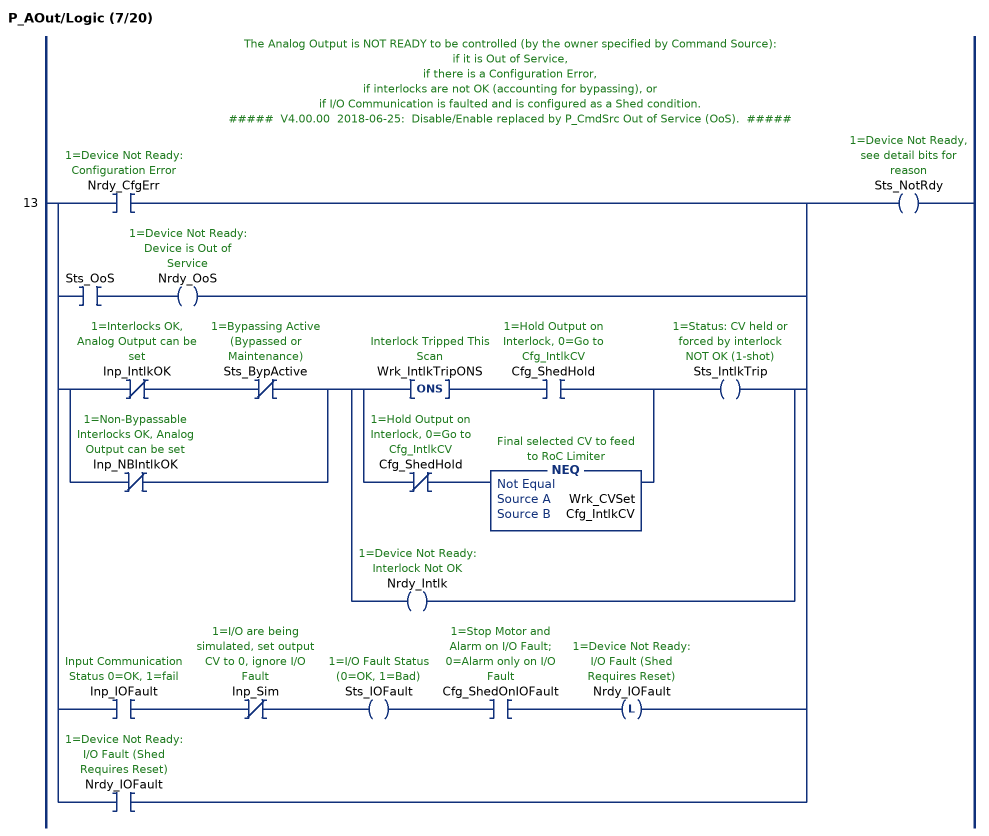
   // The Analog Output is NOT READY to be controlled (by the owner specified by Command Source):
   // if it is Out of Service,
   // if there is a Configuration Error,
   // if interlocks are not OK (accounting for bypassing), or
   // if I/O Communication is faulted and is configured as a Shed condition.
   // #####  V4.00.00  2018-06-25:  Disable/Enable replaced by P_CmdSrc Out of Service (OoS).  #####
   13: [XIC(Nrdy_CfgErr) ,XIC(Sts_OoS) OTE(Nrdy_OoS) ,[XIO(Inp_IntlkOK) XIO(Sts_BypActive) ,XIO(Inp_NBIntlkOK) ] [[ONS(Wrk_IntlkTripONS) XIC(Cfg_ShedHold) ,XIO(Cfg_ShedHold) NEQ(Wrk_CVSet,Cfg_IntlkCV) ] OTE(Sts_IntlkTrip) ,OTE(Nrdy_Intlk) ] ,XIC(Inp_IOFault) XIO(Inp_Sim) OTE(Sts_IOFault) XIC(Cfg_ShedOnIOFault) OTL(Nrdy_IOFault) ,XIC(Nrdy_IOFault) ]OTE(Sts_NotRdy);
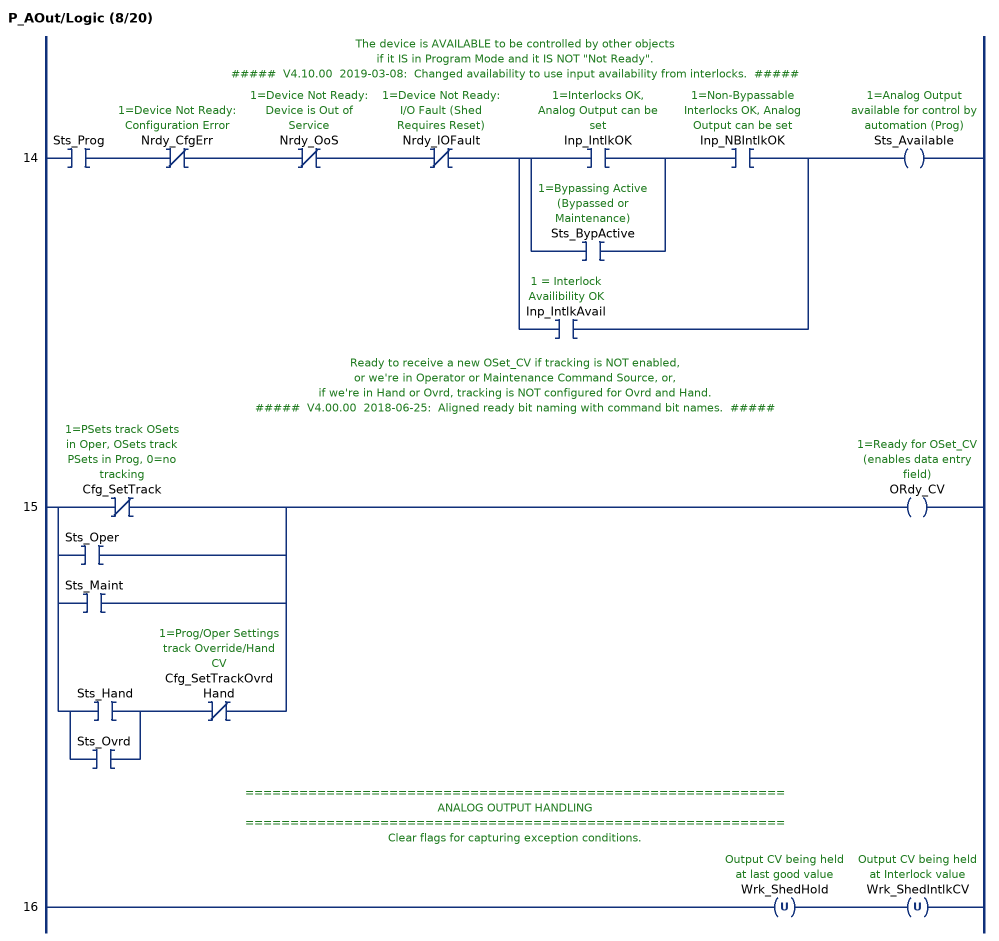
   // The device is AVAILABLE to be controlled by other objects
   // if it IS in Program Mode and it IS NOT "Not Ready".
   // #####  V4.10.00  2019-03-08:  Changed availability to use input availability from interlocks.  #####
   14: XIC(Sts_Prog)XIO(Nrdy_CfgErr)XIO(Nrdy_OoS)XIO(Nrdy_IOFault)[[XIC(Inp_IntlkOK) ,XIC(Sts_BypActive) ] XIC(Inp_NBIntlkOK) ,XIC(Inp_IntlkAvail) ]OTE(Sts_Available);
   // Ready to receive a new OSet_CV if tracking is NOT enabled,
   // or we're in Operator or Maintenance Command Source, or,
   // if we're in Hand or Ovrd, tracking is NOT configured for Ovrd and Hand.
   // #####  V4.00.00  2018-06-25:  Aligned ready bit naming with command bit names.  #####
   15: [XIO(Cfg_SetTrack) ,XIC(Sts_Oper) ,XIC(Sts_Maint) ,[XIC(Sts_Hand) ,XIC(Sts_Ovrd) ] XIO(Cfg_SetTrackOvrdHand) ]OTE(ORdy_CV);
   // ============================================================
   // ANALOG OUTPUT HANDLING
   // ============================================================
   // Clear flags for capturing exception conditions.
   16: OTU(Wrk_ShedHold)OTU(Wrk_ShedIntlkCV);
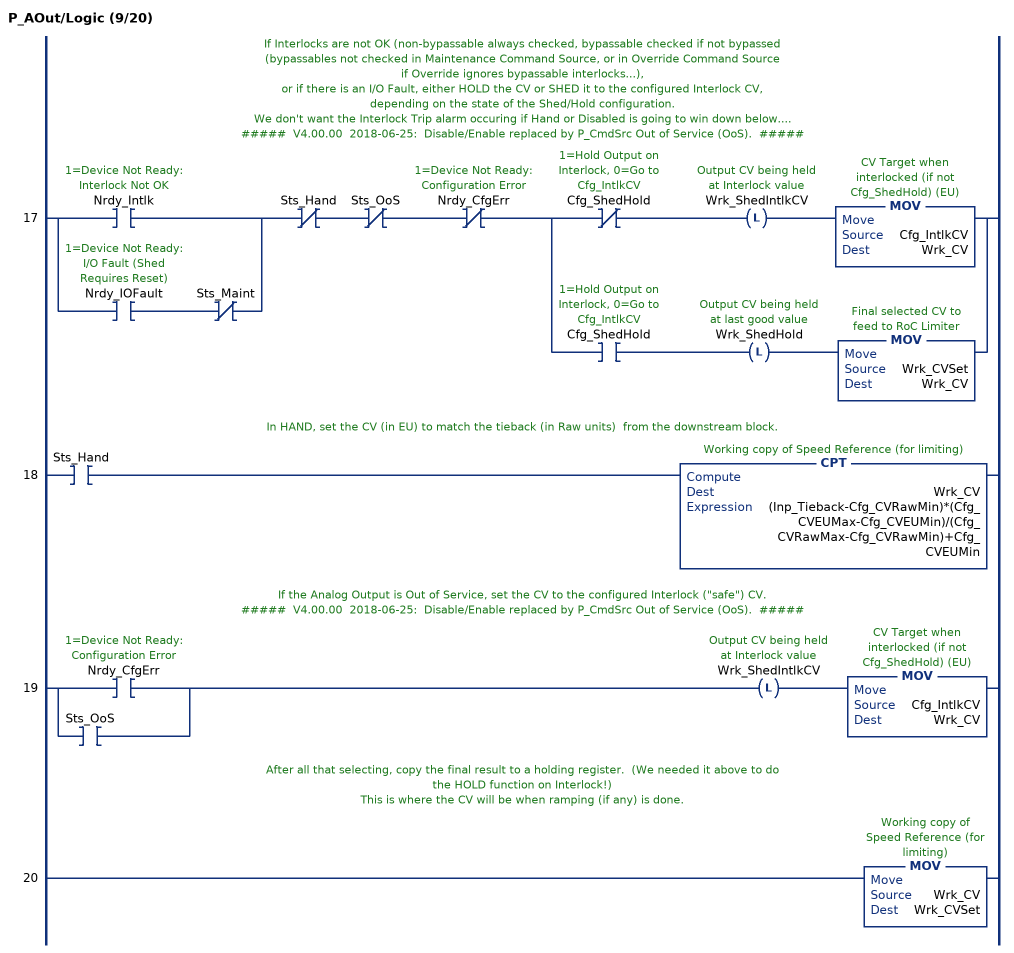
   // If Interlocks are not OK (non-bypassable always checked, bypassable checked if not bypassed
   // (bypassables not checked in Maintenance Command Source, or in Override Command Source
   //  if Override ignores bypassable interlocks...),
   // or if there is an I/O Fault, either HOLD the CV or SHED it to the configured Interlock CV,
   // depending on the state of the Shed/Hold configuration.
   // We don't want the Interlock Trip alarm occuring if Hand or Disabled is going to win down below....
   // #####  V4.00.00  2018-06-25:  Disable/Enable replaced by P_CmdSrc Out of Service (OoS).  #####
   17: [XIC(Nrdy_Intlk) ,XIC(Nrdy_IOFault) XIO(Sts_Maint) ]XIO(Sts_Hand)XIO(Sts_OoS)XIO(Nrdy_CfgErr)[XIO(Cfg_ShedHold) OTL(Wrk_ShedIntlkCV) MOV(Cfg_IntlkCV,Wrk_CV) ,XIC(Cfg_ShedHold) OTL(Wrk_ShedHold) MOV(Wrk_CVSet,Wrk_CV) ];
   // In HAND, set the CV (in EU) to match the tieback (in Raw units)  from the downstream block.
   18: XIC(Sts_Hand)CPT(Wrk_CV,(Inp_Tieback-Cfg_CVRawMin)*(Cfg_CVEUMax-Cfg_CVEUMin)/(Cfg_CVRawMax-Cfg_CVRawMin)+Cfg_CVEUMin);
   // If the Analog Output is Out of Service, set the CV to the configured Interlock ("safe") CV.
   // #####  V4.00.00  2018-06-25:  Disable/Enable replaced by P_CmdSrc Out of Service (OoS).  #####
   19: [XIC(Nrdy_CfgErr) ,XIC(Sts_OoS) ]OTL(Wrk_ShedIntlkCV)MOV(Cfg_IntlkCV,Wrk_CV);
   // After all that selecting, copy the final result to a holding register.  (We needed it above to do
   // the HOLD function on Interlock!)
   // This is where the CV will be when ramping (if any) is done.
   20: MOV(Wrk_CV,Wrk_CVSet);
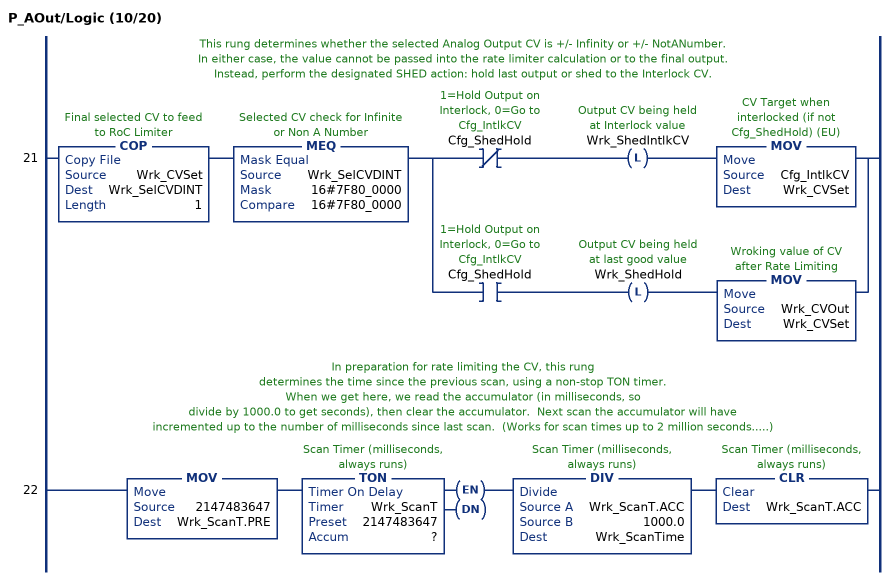
   // This rung determines whether the selected Analog Output CV is +/- Infinity or +/- NotANumber.
   // In either case, the value cannot be passed into the rate limiter calculation or to the final output.
   // Instead, perform the designated SHED action: hold last output or shed to the Interlock CV.
   21: COP(Wrk_CVSet,Wrk_SelCVDINT,1)MEQ(Wrk_SelCVDINT,16#7F80_0000,16#7F80_0000)[XIO(Cfg_ShedHold) OTL(Wrk_ShedIntlkCV) MOV(Cfg_IntlkCV,Wrk_CVSet) ,XIC(Cfg_ShedHold) OTL(Wrk_ShedHold) MOV(Wrk_CVOut,Wrk_CVSet) ];
   // In preparation for rate limiting the CV, this rung
   // determines the time since the previous scan, using a non-stop TON timer.
   // When we get here, we read the accumulator (in milliseconds, so
   // divide by 1000.0 to get seconds), then clear the accumulator.  Next scan the accumulator will have
   // incremented up to the number of milliseconds since last scan.  (Works for scan times up to 2 million seconds.....)
   22: MOV(2147483647,Wrk_ScanT.PRE)TON(Wrk_ScanT,?,?)DIV(Wrk_ScanT.ACC,1000.0,Wrk_ScanTime)CLR(Wrk_ScanT.ACC);
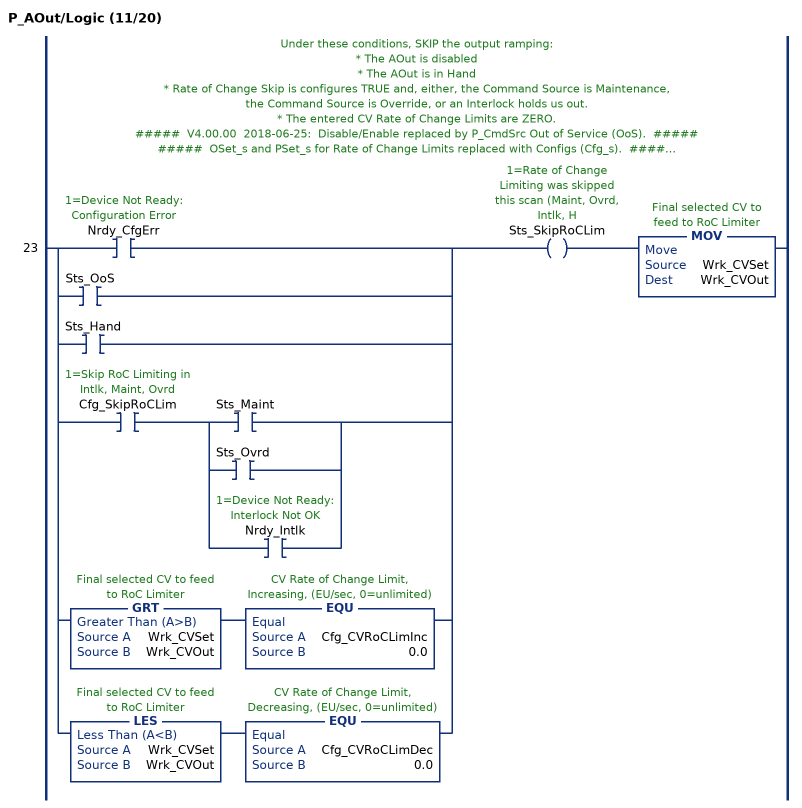
   // Under these conditions, SKIP the output ramping:
   // * The AOut is disabled
   // * The AOut is in Hand
   // * Rate of Change Skip is configures TRUE and, either, the Command Source is Maintenance,
   // the Command Source is Override, or an Interlock holds us out.
   // * The entered CV Rate of Change Limits are ZERO.
   // #####  V4.00.00  2018-06-25:  Disable/Enable replaced by P_CmdSrc Out of Service (OoS).  #####
   // #####  OSet_s and PSet_s for Rate of Change Limits replaced with Configs (Cfg_s).  #####
   // #####  Corrected CV Rate of Change Limiting when one direction is unlimited.  #####
   23: [XIC(Nrdy_CfgErr) ,XIC(Sts_OoS) ,XIC(Sts_Hand) ,XIC(Cfg_SkipRoCLim) [XIC(Sts_Maint) ,XIC(Sts_Ovrd) ,XIC(Nrdy_Intlk) ] ,GRT(Wrk_CVSet,Wrk_CVOut) EQU(Cfg_CVRoCLimInc,0.0) ,LES(Wrk_CVSet,Wrk_CVOut) EQU(Cfg_CVRoCLimDec,0.0) ]OTE(Sts_SkipRoCLim)MOV(Wrk_CVSet,Wrk_CVOut);
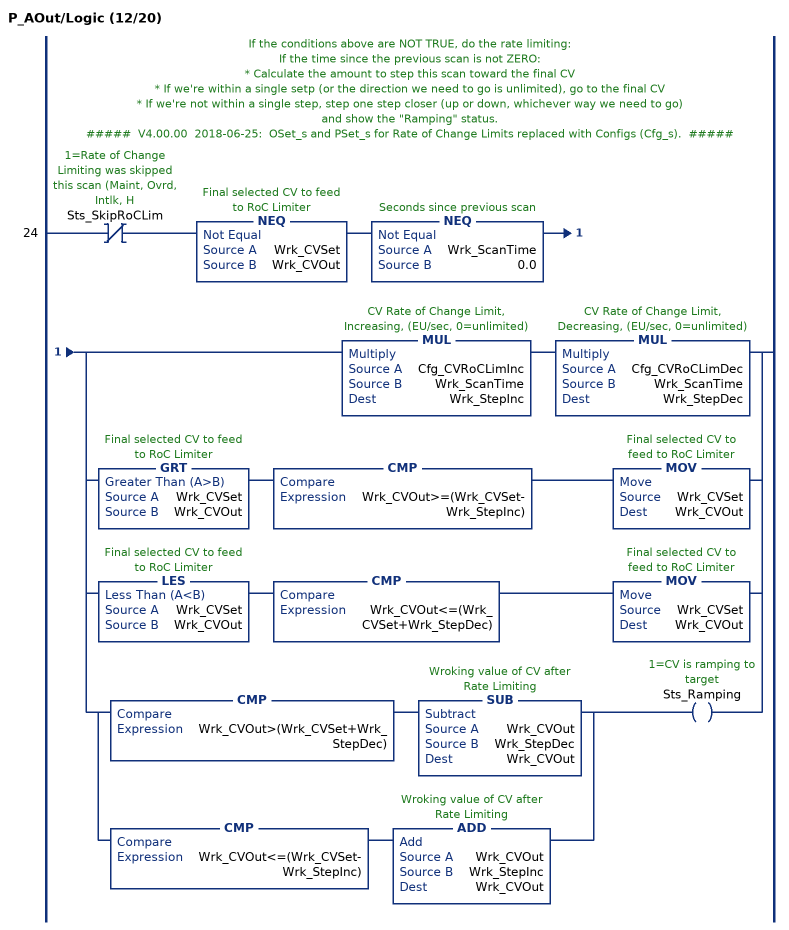
   // If the conditions above are NOT TRUE, do the rate limiting:
   // If the time since the previous scan is not ZERO:
   // * Calculate the amount to step this scan toward the final CV
   // * If we're within a single setp (or the direction we need to go is unlimited), go to the final CV
   // * If we're not within a single step, step one step closer (up or down, whichever way we need to go)
   // and show the "Ramping" status.
   // #####  V4.00.00  2018-06-25:  OSet_s and PSet_s for Rate of Change Limits replaced with Configs (Cfg_s).  #####
   24: XIO(Sts_SkipRoCLim)NEQ(Wrk_CVSet,Wrk_CVOut)NEQ(Wrk_ScanTime,0.0)[MUL(Cfg_CVRoCLimInc,Wrk_ScanTime,Wrk_StepInc) MUL(Cfg_CVRoCLimDec,Wrk_ScanTime,Wrk_StepDec) ,GRT(Wrk_CVSet,Wrk_CVOut) CMP(Wrk_CVOut>=(Wrk_CVSet-Wrk_StepInc)) MOV(Wrk_CVSet,Wrk_CVOut) ,LES(Wrk_CVSet,Wrk_CVOut) CMP(Wrk_CVOut<=(Wrk_CVSet+Wrk_StepDec)) MOV(Wrk_CVSet,Wrk_CVOut) ,[CMP(Wrk_CVOut>(Wrk_CVSet+Wrk_StepDec)) SUB(Wrk_CVOut,Wrk_StepDec,Wrk_CVOut) ,CMP(Wrk_CVOut<=(Wrk_CVSet-Wrk_StepInc)) ADD(Wrk_CVOut,Wrk_StepInc,Wrk_CVOut) ] OTE(Sts_Ramping) ];
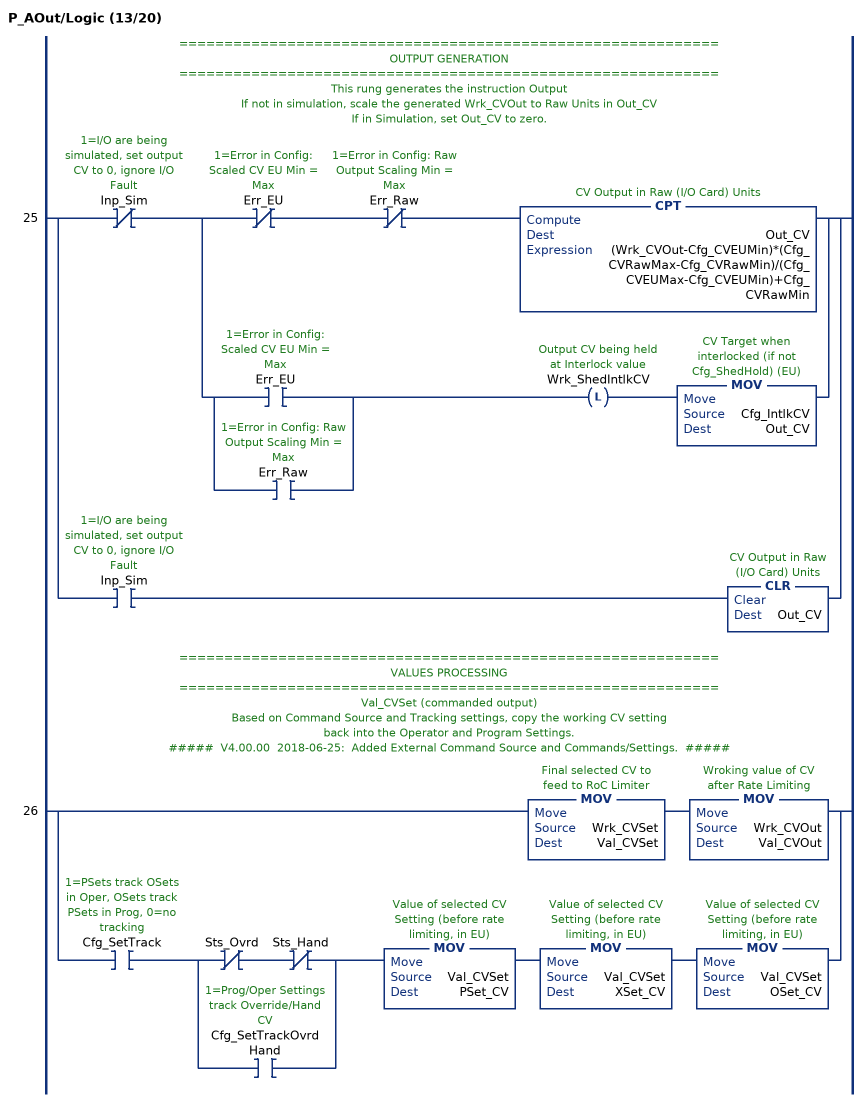
   // ============================================================
   // OUTPUT GENERATION
   // ============================================================
   // This rung generates the instruction Output
   // If not in simulation, scale the generated Wrk_CVOut to Raw Units in Out_CV
   // If in Simulation, set Out_CV to zero.
   25: [XIO(Inp_Sim) [XIO(Err_EU) XIO(Err_Raw) CPT(Out_CV,(Wrk_CVOut-Cfg_CVEUMin)*(Cfg_CVRawMax-Cfg_CVRawMin)/(Cfg_CVEUMax-Cfg_CVEUMin)+Cfg_CVRawMin) ,[XIC(Err_EU) ,XIC(Err_Raw) ] OTL(Wrk_ShedIntlkCV) MOV(Cfg_IntlkCV,Out_CV) ] ,XIC(Inp_Sim) CLR(Out_CV) ];
   // ============================================================
   // VALUES PROCESSING
   // ============================================================
   // Val_CVSet (commanded output)
   // Based on Command Source and Tracking settings, copy the working CV setting
   // back into the Operator and Program Settings.
   // #####  V4.00.00  2018-06-25:  Added External Command Source and Commands/Settings.  #####
   26: [MOV(Wrk_CVSet,Val_CVSet) MOV(Wrk_CVOut,Val_CVOut) ,XIC(Cfg_SetTrack) [XIO(Sts_Ovrd) XIO(Sts_Hand) ,XIC(Cfg_SetTrackOvrdHand) ] MOV(Val_CVSet,PSet_CV) MOV(Val_CVSet,XSet_CV) MOV(Val_CVSet,OSet_CV) ];
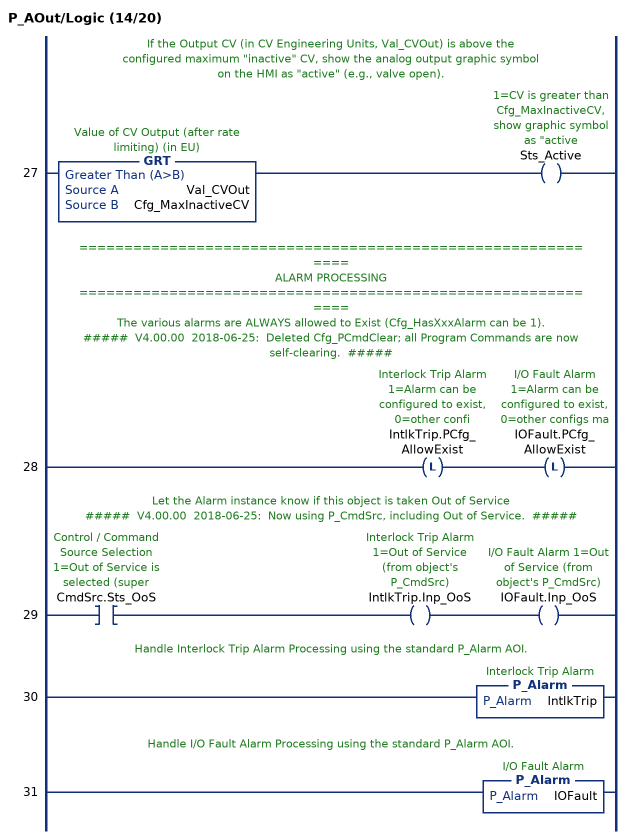
   // If the Output CV (in CV Engineering Units, Val_CVOut) is above the
   // configured maximum "inactive" CV, show the analog output graphic symbol
   // on the HMI as "active" (e.g., valve open).
   27: GRT(Val_CVOut,Cfg_MaxInactiveCV)OTE(Sts_Active);
   // ============================================================
   // ALARM PROCESSING
   // ============================================================
   // The various alarms are ALWAYS allowed to Exist (Cfg_HasXxxAlarm can be 1).
   // #####  V4.00.00  2018-06-25:  Deleted Cfg_PCmdClear; all Program Commands are now self-clearing.  #####
   28: OTL(IntlkTrip.PCfg_AllowExist)OTL(IOFault.PCfg_AllowExist);
   // Let the Alarm instance know if this object is taken Out of Service
   // #####  V4.00.00  2018-06-25:  Now using P_CmdSrc, including Out of Service.  #####
   29: XIC(CmdSrc.Sts_OoS)OTE(IntlkTrip.Inp_OoS)OTE(IOFault.Inp_OoS);
   // Handle Interlock Trip Alarm Processing using the standard P_Alarm AOI.
   30: P_Alarm(IntlkTrip);
   // Handle I/O Fault Alarm Processing using the standard P_Alarm AOI.
   31: P_Alarm(IOFault);
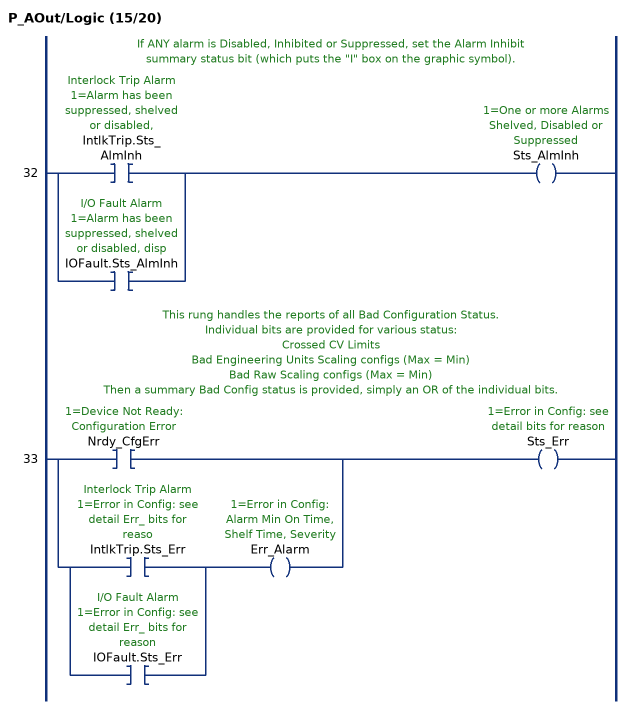
   // If ANY alarm is Disabled, Inhibited or Suppressed, set the Alarm Inhibit
   // summary status bit (which puts the "I" box on the graphic symbol).
   32: [XIC(IntlkTrip.Sts_AlmInh) ,XIC(IOFault.Sts_AlmInh) ]OTE(Sts_AlmInh);
   // This rung handles the reports of all Bad Configuration Status.
   // Individual bits are provided for various status:
   // Crossed CV Limits
   // Bad Engineering Units Scaling configs (Max = Min)
   // Bad Raw Scaling configs (Max = Min)
   // Then a summary Bad Config status is provided, simply an OR of the individual bits.
   33: [XIC(Nrdy_CfgErr) ,[XIC(IntlkTrip.Sts_Err) ,XIC(IOFault.Sts_Err) ] OTE(Err_Alarm) ]OTE(Sts_Err);
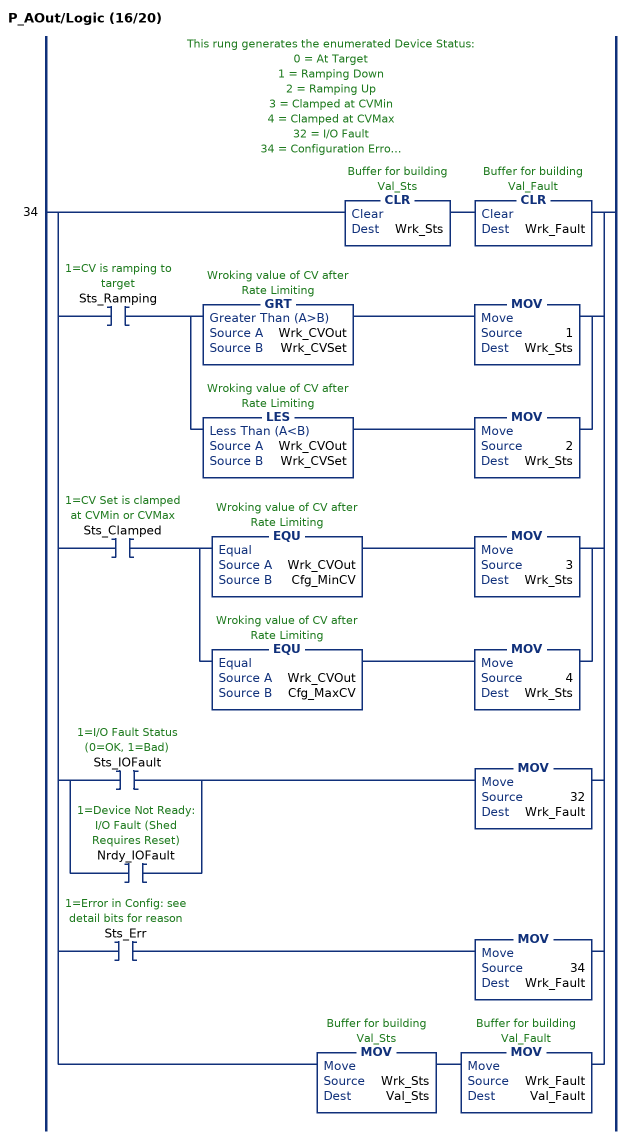
   // This rung generates the enumerated Device Status:
   // 0 = At Target
   // 1 = Ramping Down
   // 2 = Ramping Up
   // 3 = Clamped at CVMin
   // 4 = Clamped at CVMax
   // 32 = I/O Fault
   // 34 = Configuration Error
   // #####  V4.00.00  2018-06-25:  Disable/Enable replaced by P_CmdSrc Out of Service (OoS).  #####
   34: [CLR(Wrk_Sts) CLR(Wrk_Fault) ,XIC(Sts_Ramping) [GRT(Wrk_CVOut,Wrk_CVSet) MOV(1,Wrk_Sts) ,LES(Wrk_CVOut,Wrk_CVSet) MOV(2,Wrk_Sts) ] ,XIC(Sts_Clamped) [EQU(Wrk_CVOut,Cfg_MinCV) MOV(3,Wrk_Sts) ,EQU(Wrk_CVOut,Cfg_MaxCV) MOV(4,Wrk_Sts) ] ,[XIC(Sts_IOFault) ,XIC(Nrdy_IOFault) ] MOV(32,Wrk_Fault) ,XIC(Sts_Err) MOV(34,Wrk_Fault) ,MOV(Wrk_Sts,Val_Sts) MOV(Wrk_Fault,Val_Fault) ];
